  PROC DrawPart176()
    MoveL Offs(pOrigin,258.82,201.40,0.00),v40,fine,tPen\WObj:=wPaper;
    MoveL Offs(pOrigin,258.82,201.40,6.00),v60,z5,tPen\WObj:=wPaper;
    MoveL Offs(pOrigin,257.32,201.40,6.00),vTravel,z5,tPen\WObj:=wPaper;
    MoveL Offs(pOrigin,257.32,201.40,0.00),v60,z0,tPen\WObj:=wPaper;
    MoveL Offs(pOrigin,259.12,199.60,0.00),v40,fine,tPen\WObj:=wPaper;
    MoveL Offs(pOrigin,259.12,199.60,6.00),v60,z5,tPen\WObj:=wPaper;
    MoveL Offs(pOrigin,257.63,199.61,6.00),vTravel,z5,tPen\WObj:=wPaper;
    MoveL Offs(pOrigin,257.63,199.61,0.00),v60,z0,tPen\WObj:=wPaper;
    MoveL Offs(pOrigin,255.52,201.71,0.00),v40,fine,tPen\WObj:=wPaper;
    MoveL Offs(pOrigin,255.52,201.71,6.00),v60,z5,tPen\WObj:=wPaper;
    MoveL Offs(pOrigin,253.72,202.01,6.00),vTravel,z5,tPen\WObj:=wPaper;
    MoveL Offs(pOrigin,253.72,202.01,0.00),v60,z0,tPen\WObj:=wPaper;
    MoveL Offs(pOrigin,255.98,199.76,0.00),v40,fine,tPen\WObj:=wPaper;
    MoveL Offs(pOrigin,255.98,199.76,6.00),v60,z5,tPen\WObj:=wPaper;
    MoveL Offs(pOrigin,254.48,199.77,6.00),vTravel,z5,tPen\WObj:=wPaper;
    MoveL Offs(pOrigin,254.48,199.77,0.00),v60,z0,tPen\WObj:=wPaper;
    MoveL Offs(pOrigin,252.23,202.02,0.00),v40,z0,tPen\WObj:=wPaper;
    MoveL Offs(pOrigin,251.94,201.46,0.00),v40,z0,tPen\WObj:=wPaper;
    MoveL Offs(pOrigin,251.19,200.71,0.00),v40,z0,tPen\WObj:=wPaper;
    MoveL Offs(pOrigin,251.33,199.92,0.00),v40,z0,tPen\WObj:=wPaper;
    MoveL Offs(pOrigin,249.53,201.73,0.00),v40,fine,tPen\WObj:=wPaper;
    MoveL Offs(pOrigin,249.53,201.73,6.00),v60,z5,tPen\WObj:=wPaper;
    MoveL Offs(pOrigin,250.73,202.02,6.00),vTravel,z5,tPen\WObj:=wPaper;
    MoveL Offs(pOrigin,250.73,202.02,0.00),v60,z0,tPen\WObj:=wPaper;
    MoveL Offs(pOrigin,252.98,199.77,0.00),v40,fine,tPen\WObj:=wPaper;
    MoveL Offs(pOrigin,252.98,199.77,6.00),v60,z5,tPen\WObj:=wPaper;
    MoveL Offs(pOrigin,251.76,206.96,6.00),vTravel,z5,tPen\WObj:=wPaper;
    MoveL Offs(pOrigin,251.76,206.96,0.00),v60,z0,tPen\WObj:=wPaper;
    MoveL Offs(pOrigin,249.06,209.67,0.00),v40,z0,tPen\WObj:=wPaper;
    MoveL Offs(pOrigin,249.42,209.39,0.00),v40,z0,tPen\WObj:=wPaper;
    MoveL Offs(pOrigin,247.16,207.14,0.00),v40,z0,tPen\WObj:=wPaper;
    MoveL Offs(pOrigin,247.57,206.68,0.00),v40,z0,tPen\WObj:=wPaper;
    MoveL Offs(pOrigin,245.01,209.23,0.00),v40,z0,tPen\WObj:=wPaper;
    MoveL Offs(pOrigin,244.47,208.93,0.00),v40,z0,tPen\WObj:=wPaper;
    MoveL Offs(pOrigin,242.67,207.12,0.00),v40,z0,tPen\WObj:=wPaper;
    MoveL Offs(pOrigin,243.07,206.69,0.00),v40,z0,tPen\WObj:=wPaper;
    MoveL Offs(pOrigin,240.37,209.40,0.00),v40,z0,tPen\WObj:=wPaper;
    MoveL Offs(pOrigin,239.98,208.91,0.00),v40,z0,tPen\WObj:=wPaper;
    MoveL Offs(pOrigin,238.78,207.71,0.00),v40,z0,tPen\WObj:=wPaper;
    MoveL Offs(pOrigin,238.10,208.15,0.00),v40,z0,tPen\WObj:=wPaper;
    MoveL Offs(pOrigin,240.86,207.51,0.00),v40,z0,tPen\WObj:=wPaper;
    MoveL Offs(pOrigin,248.30,207.51,0.00),v40,z0,tPen\WObj:=wPaper;
    MoveL Offs(pOrigin,256.16,208.79,0.00),v40,z0,tPen\WObj:=wPaper;
    MoveL Offs(pOrigin,259.14,209.71,0.00),v40,z0,tPen\WObj:=wPaper;
    MoveL Offs(pOrigin,259.56,210.49,0.00),v40,z0,tPen\WObj:=wPaper;
    MoveL Offs(pOrigin,259.56,210.49,0.00),v40,z0,tPen\WObj:=wPaper;
    MoveL Offs(pOrigin,253.61,209.21,0.00),v40,z0,tPen\WObj:=wPaper;
    MoveL Offs(pOrigin,247.24,208.36,0.00),v40,z0,tPen\WObj:=wPaper;
    MoveL Offs(pOrigin,241.07,208.36,0.00),v40,z0,tPen\WObj:=wPaper;
    MoveL Offs(pOrigin,238.10,208.79,0.00),v40,z0,tPen\WObj:=wPaper;
    MoveL Offs(pOrigin,238.10,208.79,0.00),v40,z0,tPen\WObj:=wPaper;
    MoveL Offs(pOrigin,237.04,209.00,0.00),v40,z0,tPen\WObj:=wPaper;
    MoveL Offs(pOrigin,237.04,209.00,0.00),v40,z0,tPen\WObj:=wPaper;
    MoveL Offs(pOrigin,237.46,208.15,0.00),v40,z0,tPen\WObj:=wPaper;
    MoveL Offs(pOrigin,237.89,208.15,0.00),v40,z0,tPen\WObj:=wPaper;
    MoveL Offs(pOrigin,238.10,208.79,0.00),v40,z0,tPen\WObj:=wPaper;
    MoveL Offs(pOrigin,238.63,209.06,0.00),v40,z0,tPen\WObj:=wPaper;
    MoveL Offs(pOrigin,237.58,208.01,0.00),v40,z0,tPen\WObj:=wPaper;
    MoveL Offs(pOrigin,237.04,209.00,0.00),v40,z0,tPen\WObj:=wPaper;
    MoveL Offs(pOrigin,234.49,209.35,0.00),v40,z0,tPen\WObj:=wPaper;
    MoveL Offs(pOrigin,232.15,210.70,0.00),v40,z0,tPen\WObj:=wPaper;
    MoveL Offs(pOrigin,231.51,210.91,0.00),v40,z0,tPen\WObj:=wPaper;
    MoveL Offs(pOrigin,230.45,212.12,0.00),v40,z0,tPen\WObj:=wPaper;
    MoveL Offs(pOrigin,227.26,214.52,0.00),v40,fine,tPen\WObj:=wPaper;
    MoveL Offs(pOrigin,227.26,214.52,6.00),v60,z5,tPen\WObj:=wPaper;
    MoveL Offs(pOrigin,228.97,213.33,6.00),vTravel,z5,tPen\WObj:=wPaper;
    MoveL Offs(pOrigin,228.97,213.33,0.00),v60,z0,tPen\WObj:=wPaper;
    MoveL Offs(pOrigin,234.08,208.22,0.00),v40,z0,tPen\WObj:=wPaper;
    MoveL Offs(pOrigin,234.29,209.19,0.00),v40,z0,tPen\WObj:=wPaper;
    MoveL Offs(pOrigin,235.04,209.94,0.00),v40,z0,tPen\WObj:=wPaper;
    MoveL Offs(pOrigin,233.99,210.39,0.00),v40,z0,tPen\WObj:=wPaper;
    MoveL Offs(pOrigin,233.24,209.64,0.00),v40,fine,tPen\WObj:=wPaper;
    MoveL Offs(pOrigin,233.24,209.64,6.00),v60,z5,tPen\WObj:=wPaper;
    MoveL Offs(pOrigin,234.07,211.21,6.00),vTravel,z5,tPen\WObj:=wPaper;
    MoveL Offs(pOrigin,234.07,211.21,0.00),v60,z0,tPen\WObj:=wPaper;
    MoveL Offs(pOrigin,238.28,207.01,0.00),v40,fine,tPen\WObj:=wPaper;
    MoveL Offs(pOrigin,238.28,207.01,6.00),v60,z5,tPen\WObj:=wPaper;
    MoveL Offs(pOrigin,239.93,206.85,6.00),vTravel,z5,tPen\WObj:=wPaper;
    MoveL Offs(pOrigin,239.93,206.85,0.00),v60,z0,tPen\WObj:=wPaper;
    MoveL Offs(pOrigin,236.47,210.31,0.00),v40,z0,tPen\WObj:=wPaper;
    MoveL Offs(pOrigin,236.39,209.80,0.00),v40,z0,tPen\WObj:=wPaper;
    MoveL Offs(pOrigin,235.19,208.60,0.00),v40,z0,tPen\WObj:=wPaper;
    MoveL Offs(pOrigin,236.23,208.15,0.00),v40,z0,tPen\WObj:=wPaper;
    MoveL Offs(pOrigin,237.43,209.35,0.00),v40,z0,tPen\WObj:=wPaper;
    MoveL Offs(pOrigin,238.57,209.70,0.00),v40,z0,tPen\WObj:=wPaper;
    MoveL Offs(pOrigin,241.58,206.70,0.00),v40,z0,tPen\WObj:=wPaper;
    MoveL Offs(pOrigin,241.47,207.42,0.00),v40,z0,tPen\WObj:=wPaper;
    MoveL Offs(pOrigin,242.98,208.92,0.00),v40,z0,tPen\WObj:=wPaper;
    MoveL Offs(pOrigin,243.52,209.24,0.00),v40,z0,tPen\WObj:=wPaper;
    MoveL Offs(pOrigin,246.07,206.68,0.00),v40,z0,tPen\WObj:=wPaper;
    MoveL Offs(pOrigin,245.67,207.13,0.00),v40,z0,tPen\WObj:=wPaper;
    MoveL Offs(pOrigin,247.62,209.08,0.00),v40,z0,tPen\WObj:=wPaper;
    MoveL Offs(pOrigin,247.86,209.37,0.00),v40,z0,tPen\WObj:=wPaper;
    MoveL Offs(pOrigin,250.41,206.82,0.00),v40,z0,tPen\WObj:=wPaper;
    MoveL Offs(pOrigin,250.61,207.60,0.00),v40,z0,tPen\WObj:=wPaper;
    MoveL Offs(pOrigin,252.87,209.85,0.00),v40,z0,tPen\WObj:=wPaper;
    MoveL Offs(pOrigin,253.10,210.11,0.00),v40,z0,tPen\WObj:=wPaper;
    MoveL Offs(pOrigin,255.50,207.70,0.00),v40,z0,tPen\WObj:=wPaper;
    MoveL Offs(pOrigin,255.86,208.36,0.00),v40,z0,tPen\WObj:=wPaper;
    MoveL Offs(pOrigin,258.26,210.77,0.00),v40,z0,tPen\WObj:=wPaper;
    MoveL Offs(pOrigin,258.04,211.14,0.00),v40,z0,tPen\WObj:=wPaper;
    MoveL Offs(pOrigin,260.14,209.04,0.00),v40,z0,tPen\WObj:=wPaper;
    MoveL Offs(pOrigin,260.06,209.57,0.00),v40,z0,tPen\WObj:=wPaper;
    MoveL Offs(pOrigin,263.36,212.88,0.00),v40,z0,tPen\WObj:=wPaper;
    MoveL Offs(pOrigin,263.28,213.37,0.00),v40,z0,tPen\WObj:=wPaper;
    MoveL Offs(pOrigin,265.08,211.57,0.00),v40,z0,tPen\WObj:=wPaper;
    MoveL Offs(pOrigin,264.45,212.40,0.00),v40,z0,tPen\WObj:=wPaper;
    MoveL Offs(pOrigin,265.73,212.19,0.00),v40,z0,tPen\WObj:=wPaper;
    MoveL Offs(pOrigin,265.94,212.82,0.00),v40,z0,tPen\WObj:=wPaper;
    MoveL Offs(pOrigin,265.83,212.31,0.00),v40,z0,tPen\WObj:=wPaper;
    MoveL Offs(pOrigin,264.32,213.82,0.00),v40,z0,tPen\WObj:=wPaper;
    MoveL Offs(pOrigin,265.22,214.41,0.00),v40,z0,tPen\WObj:=wPaper;
    MoveL Offs(pOrigin,266.72,212.91,0.00),v40,z0,tPen\WObj:=wPaper;
    MoveL Offs(pOrigin,267.32,213.81,0.00),v40,z0,tPen\WObj:=wPaper;
    MoveL Offs(pOrigin,265.97,215.16,0.00),v40,z0,tPen\WObj:=wPaper;
    MoveL Offs(pOrigin,266.36,214.39,0.00),v40,z0,tPen\WObj:=wPaper;
    MoveL Offs(pOrigin,262.60,210.63,0.00),v40,z0,tPen\WObj:=wPaper;
    MoveL Offs(pOrigin,263.29,210.37,0.00),v40,z0,tPen\WObj:=wPaper;
    MoveL Offs(pOrigin,261.33,212.33,0.00),v40,z0,tPen\WObj:=wPaper;
    MoveL Offs(pOrigin,262.38,212.77,0.00),v40,z0,tPen\WObj:=wPaper;
  ENDPROC

  PROC DrawPart177()
    MoveL Offs(pOrigin,264.18,210.97,0.00),v40,fine,tPen\WObj:=wPaper;
    MoveL Offs(pOrigin,264.18,210.97,6.00),v60,z5,tPen\WObj:=wPaper;
    MoveL Offs(pOrigin,264.45,212.40,6.00),vTravel,z5,tPen\WObj:=wPaper;
    MoveL Offs(pOrigin,264.45,212.40,0.00),v60,z0,tPen\WObj:=wPaper;
    MoveL Offs(pOrigin,262.33,211.20,0.00),v40,z0,tPen\WObj:=wPaper;
    MoveL Offs(pOrigin,259.56,210.49,0.00),v40,z0,tPen\WObj:=wPaper;
    MoveL Offs(pOrigin,259.24,211.44,0.00),v40,z0,tPen\WObj:=wPaper;
    MoveL Offs(pOrigin,261.19,209.48,0.00),v40,z0,tPen\WObj:=wPaper;
    MoveL Offs(pOrigin,262.24,209.93,0.00),v40,z0,tPen\WObj:=wPaper;
    MoveL Offs(pOrigin,260.29,211.88,0.00),v40,z0,tPen\WObj:=wPaper;
    MoveL Offs(pOrigin,260.36,211.37,0.00),v40,z0,tPen\WObj:=wPaper;
    MoveL Offs(pOrigin,257.96,208.97,0.00),v40,z0,tPen\WObj:=wPaper;
    MoveL Offs(pOrigin,257.90,208.29,0.00),v40,z0,tPen\WObj:=wPaper;
    MoveL Offs(pOrigin,255.65,210.55,0.00),v40,z0,tPen\WObj:=wPaper;
    MoveL Offs(pOrigin,256.46,210.46,0.00),v40,z0,tPen\WObj:=wPaper;
    MoveL Offs(pOrigin,254.21,208.21,0.00),v40,z0,tPen\WObj:=wPaper;
    MoveL Offs(pOrigin,254.31,207.41,0.00),v40,z0,tPen\WObj:=wPaper;
    MoveL Offs(pOrigin,251.60,210.11,0.00),v40,z0,tPen\WObj:=wPaper;
    MoveL Offs(pOrigin,251.07,209.54,0.00),v40,z0,tPen\WObj:=wPaper;
    MoveL Offs(pOrigin,248.96,207.44,0.00),v40,z0,tPen\WObj:=wPaper;
    MoveL Offs(pOrigin,248.92,206.82,0.00),v40,z0,tPen\WObj:=wPaper;
    MoveL Offs(pOrigin,246.51,209.23,0.00),v40,z0,tPen\WObj:=wPaper;
    MoveL Offs(pOrigin,245.97,208.93,0.00),v40,z0,tPen\WObj:=wPaper;
    MoveL Offs(pOrigin,244.17,207.13,0.00),v40,z0,tPen\WObj:=wPaper;
    MoveL Offs(pOrigin,244.57,206.69,0.00),v40,z0,tPen\WObj:=wPaper;
    MoveL Offs(pOrigin,242.02,209.24,0.00),v40,z0,tPen\WObj:=wPaper;
    MoveL Offs(pOrigin,241.48,208.92,0.00),v40,z0,tPen\WObj:=wPaper;
    MoveL Offs(pOrigin,240.13,207.56,0.00),v40,fine,tPen\WObj:=wPaper;
    MoveL Offs(pOrigin,240.13,207.56,6.00),v60,z5,tPen\WObj:=wPaper;
    MoveL Offs(pOrigin,236.48,207.31,6.00),vTravel,z5,tPen\WObj:=wPaper;
    MoveL Offs(pOrigin,236.48,207.31,0.00),v60,z0,tPen\WObj:=wPaper;
    MoveL Offs(pOrigin,231.22,212.57,0.00),v40,fine,tPen\WObj:=wPaper;
    MoveL Offs(pOrigin,231.22,212.57,6.00),v60,z5,tPen\WObj:=wPaper;
    MoveL Offs(pOrigin,229.60,208.36,6.00),vTravel,z5,tPen\WObj:=wPaper;
    MoveL Offs(pOrigin,229.60,208.36,0.00),v60,z0,tPen\WObj:=wPaper;
    MoveL Offs(pOrigin,227.90,208.72,0.00),v40,z0,tPen\WObj:=wPaper;
    MoveL Offs(pOrigin,222.16,210.98,0.00),v40,z0,tPen\WObj:=wPaper;
    MoveL Offs(pOrigin,215.15,217.29,0.00),v40,z0,tPen\WObj:=wPaper;
    MoveL Offs(pOrigin,211.89,221.75,0.00),v40,z0,tPen\WObj:=wPaper;
    MoveL Offs(pOrigin,209.98,225.57,0.00),v40,z0,tPen\WObj:=wPaper;
    MoveL Offs(pOrigin,207.93,232.38,0.00),v40,z0,tPen\WObj:=wPaper;
    MoveL Offs(pOrigin,207.29,232.38,0.00),v40,z0,tPen\WObj:=wPaper;
    MoveL Offs(pOrigin,207.07,233.44,0.00),v40,z0,tPen\WObj:=wPaper;
    MoveL Offs(pOrigin,207.29,233.65,0.00),v40,z0,tPen\WObj:=wPaper;
    MoveL Offs(pOrigin,206.29,233.02,0.00),v40,z0,tPen\WObj:=wPaper;
    MoveL Offs(pOrigin,209.30,230.01,0.00),v40,z0,tPen\WObj:=wPaper;
    MoveL Offs(pOrigin,208.74,229.94,0.00),v40,z0,tPen\WObj:=wPaper;
    MoveL Offs(pOrigin,205.73,226.93,0.00),v40,z0,tPen\WObj:=wPaper;
    MoveL Offs(pOrigin,206.01,227.26,0.00),v40,z0,tPen\WObj:=wPaper;
    MoveL Offs(pOrigin,209.20,227.26,0.00),v40,z0,tPen\WObj:=wPaper;
    MoveL Offs(pOrigin,209.92,226.65,0.00),v40,z0,tPen\WObj:=wPaper;
    MoveL Offs(pOrigin,208.42,225.14,0.00),v40,z0,tPen\WObj:=wPaper;
    MoveL Offs(pOrigin,208.99,225.14,0.00),v40,z0,tPen\WObj:=wPaper;
    MoveL Offs(pOrigin,210.05,225.14,0.00),v40,z0,tPen\WObj:=wPaper;
    MoveL Offs(pOrigin,209.62,226.20,0.00),v40,z0,tPen\WObj:=wPaper;
    MoveL Offs(pOrigin,208.56,226.20,0.00),v40,z0,tPen\WObj:=wPaper;
    MoveL Offs(pOrigin,208.05,227.28,0.00),v40,z0,tPen\WObj:=wPaper;
    MoveL Offs(pOrigin,208.05,228.34,0.00),v40,fine,tPen\WObj:=wPaper;
    MoveL Offs(pOrigin,208.05,228.34,6.00),v60,z5,tPen\WObj:=wPaper;
    MoveL Offs(pOrigin,205.71,226.13,6.00),vTravel,z5,tPen\WObj:=wPaper;
    MoveL Offs(pOrigin,205.71,226.13,0.00),v60,z0,tPen\WObj:=wPaper;
    MoveL Offs(pOrigin,201.81,230.04,0.00),v40,z0,tPen\WObj:=wPaper;
    MoveL Offs(pOrigin,202.74,229.92,0.00),v40,z0,tPen\WObj:=wPaper;
    MoveL Offs(pOrigin,204.25,231.42,0.00),v40,z0,tPen\WObj:=wPaper;
    MoveL Offs(pOrigin,204.65,231.68,0.00),v40,z0,tPen\WObj:=wPaper;
    MoveL Offs(pOrigin,201.19,235.13,0.00),v40,z0,tPen\WObj:=wPaper;
    MoveL Offs(pOrigin,202.19,234.65,0.00),v40,z0,tPen\WObj:=wPaper;
    MoveL Offs(pOrigin,203.46,234.65,0.00),v40,z0,tPen\WObj:=wPaper;
    MoveL Offs(pOrigin,203.81,233.97,0.00),v40,z0,tPen\WObj:=wPaper;
    MoveL Offs(pOrigin,201.85,232.01,0.00),v40,z0,tPen\WObj:=wPaper;
    MoveL Offs(pOrigin,201.76,232.54,0.00),v40,z0,tPen\WObj:=wPaper;
    MoveL Offs(pOrigin,203.46,232.54,0.00),v40,z0,tPen\WObj:=wPaper;
    MoveL Offs(pOrigin,202.77,232.80,0.00),v40,z0,tPen\WObj:=wPaper;
    MoveL Offs(pOrigin,202.77,234.08,0.00),v40,z0,tPen\WObj:=wPaper;
    MoveL Offs(pOrigin,203.46,233.59,0.00),v40,z0,tPen\WObj:=wPaper;
    MoveL Offs(pOrigin,201.34,233.59,0.00),v40,fine,tPen\WObj:=wPaper;
    MoveL Offs(pOrigin,201.34,233.59,6.00),v60,z5,tPen\WObj:=wPaper;
    MoveL Offs(pOrigin,200.52,238.15,6.00),vTravel,z5,tPen\WObj:=wPaper;
    MoveL Offs(pOrigin,200.52,238.15,0.00),v60,z0,tPen\WObj:=wPaper;
    MoveL Offs(pOrigin,203.08,240.71,0.00),v40,z0,tPen\WObj:=wPaper;
    MoveL Offs(pOrigin,202.61,239.93,0.00),v40,z0,tPen\WObj:=wPaper;
    MoveL Offs(pOrigin,200.06,239.93,0.00),v40,fine,tPen\WObj:=wPaper;
    MoveL Offs(pOrigin,200.06,239.93,6.00),v60,z5,tPen\WObj:=wPaper;
    MoveL Offs(pOrigin,199.34,244.44,6.00),vTravel,z5,tPen\WObj:=wPaper;
    MoveL Offs(pOrigin,199.34,244.44,0.00),v60,z0,tPen\WObj:=wPaper;
    MoveL Offs(pOrigin,201.00,246.09,0.00),v40,fine,tPen\WObj:=wPaper;
    MoveL Offs(pOrigin,201.00,246.09,6.00),v60,z5,tPen\WObj:=wPaper;
    MoveL Offs(pOrigin,202.80,246.96,6.00),vTravel,z5,tPen\WObj:=wPaper;
    MoveL Offs(pOrigin,202.80,246.96,0.00),v60,z0,tPen\WObj:=wPaper;
    MoveL Offs(pOrigin,194.24,255.53,0.00),v40,z0,tPen\WObj:=wPaper;
    MoveL Offs(pOrigin,194.59,256.11,0.00),v40,z0,tPen\WObj:=wPaper;
    MoveL Offs(pOrigin,196.39,257.91,0.00),v40,fine,tPen\WObj:=wPaper;
    MoveL Offs(pOrigin,196.39,257.91,6.00),v60,z5,tPen\WObj:=wPaper;
    MoveL Offs(pOrigin,196.38,256.41,6.00),vTravel,z5,tPen\WObj:=wPaper;
    MoveL Offs(pOrigin,196.38,256.41,0.00),v60,z0,tPen\WObj:=wPaper;
    MoveL Offs(pOrigin,194.58,254.61,0.00),v40,z0,tPen\WObj:=wPaper;
    MoveL Offs(pOrigin,194.24,254.03,0.00),v40,z0,tPen\WObj:=wPaper;
    MoveL Offs(pOrigin,207.47,240.80,0.00),v40,z0,tPen\WObj:=wPaper;
    MoveL Offs(pOrigin,206.65,241.51,0.00),v40,z0,tPen\WObj:=wPaper;
    MoveL Offs(pOrigin,206.86,242.79,0.00),v40,z0,tPen\WObj:=wPaper;
    MoveL Offs(pOrigin,206.44,243.21,0.00),v40,z0,tPen\WObj:=wPaper;
    MoveL Offs(pOrigin,206.44,243.21,0.00),v40,z0,tPen\WObj:=wPaper;
    MoveL Offs(pOrigin,206.86,245.98,0.00),v40,z0,tPen\WObj:=wPaper;
    MoveL Offs(pOrigin,206.65,248.10,0.00),v40,z0,tPen\WObj:=wPaper;
    MoveL Offs(pOrigin,207.14,247.76,0.00),v40,z0,tPen\WObj:=wPaper;
    MoveL Offs(pOrigin,206.39,247.01,0.00),v40,fine,tPen\WObj:=wPaper;
    MoveL Offs(pOrigin,206.39,247.01,6.00),v60,z5,tPen\WObj:=wPaper;
    MoveL Offs(pOrigin,207.75,246.50,6.00),vTravel,z5,tPen\WObj:=wPaper;
    MoveL Offs(pOrigin,207.75,246.50,0.00),v60,z0,tPen\WObj:=wPaper;
    MoveL Offs(pOrigin,204.29,249.95,0.00),v40,z0,tPen\WObj:=wPaper;
    MoveL Offs(pOrigin,204.90,250.00,0.00),v40,z0,tPen\WObj:=wPaper;
    MoveL Offs(pOrigin,207.31,252.40,0.00),v40,z0,tPen\WObj:=wPaper;
    MoveL Offs(pOrigin,206.86,252.60,0.00),v40,z0,tPen\WObj:=wPaper;
    MoveL Offs(pOrigin,204.52,252.60,0.00),v40,z0,tPen\WObj:=wPaper;
    MoveL Offs(pOrigin,204.31,252.39,0.00),v40,z0,tPen\WObj:=wPaper;
    MoveL Offs(pOrigin,208.37,256.45,0.00),v40,z0,tPen\WObj:=wPaper;
    MoveL Offs(pOrigin,208.91,257.28,0.00),v40,z0,tPen\WObj:=wPaper;
    MoveL Offs(pOrigin,195.69,270.50,0.00),v40,z0,tPen\WObj:=wPaper;
    MoveL Offs(pOrigin,196.45,270.41,0.00),v40,z0,tPen\WObj:=wPaper;
    MoveL Offs(pOrigin,196.24,270.84,0.00),v40,z0,tPen\WObj:=wPaper;
  ENDPROC

  PROC DrawPart178()
    MoveL Offs(pOrigin,196.45,270.41,0.00),v40,z0,tPen\WObj:=wPaper;
    MoveL Offs(pOrigin,196.73,270.20,0.00),v40,z0,tPen\WObj:=wPaper;
    MoveL Offs(pOrigin,204.54,278.01,0.00),v40,z0,tPen\WObj:=wPaper;
    MoveL Offs(pOrigin,205.55,278.56,0.00),v40,z0,tPen\WObj:=wPaper;
    MoveL Offs(pOrigin,189.03,295.09,0.00),v40,z0,tPen\WObj:=wPaper;
    MoveL Offs(pOrigin,189.91,294.74,0.00),v40,z0,tPen\WObj:=wPaper;
    MoveL Offs(pOrigin,197.57,302.41,0.00),v40,z0,tPen\WObj:=wPaper;
    MoveL Offs(pOrigin,198.36,302.50,0.00),v40,z0,tPen\WObj:=wPaper;
    MoveL Offs(pOrigin,198.79,302.36,0.00),v40,z0,tPen\WObj:=wPaper;
    MoveL Offs(pOrigin,200.70,303.14,0.00),v40,z0,tPen\WObj:=wPaper;
    MoveL Offs(pOrigin,201.34,302.92,0.00),v40,z0,tPen\WObj:=wPaper;
    MoveL Offs(pOrigin,200.72,302.57,0.00),v40,z0,tPen\WObj:=wPaper;
    MoveL Offs(pOrigin,210.04,311.88,0.00),v40,z0,tPen\WObj:=wPaper;
    MoveL Offs(pOrigin,210.26,311.85,0.00),v40,z0,tPen\WObj:=wPaper;
    MoveL Offs(pOrigin,210.05,312.06,0.00),v40,z0,tPen\WObj:=wPaper;
    MoveL Offs(pOrigin,210.69,311.42,0.00),v40,z0,tPen\WObj:=wPaper;
    MoveL Offs(pOrigin,211.75,311.42,0.00),v40,z0,tPen\WObj:=wPaper;
    MoveL Offs(pOrigin,212.60,311.74,0.00),v40,z0,tPen\WObj:=wPaper;
    MoveL Offs(pOrigin,226.84,311.74,0.00),v40,z0,tPen\WObj:=wPaper;
    MoveL Offs(pOrigin,226.84,312.79,0.00),v40,z0,tPen\WObj:=wPaper;
    MoveL Offs(pOrigin,225.14,312.79,0.00),v40,z0,tPen\WObj:=wPaper;
    MoveL Offs(pOrigin,224.50,312.91,0.00),v40,z0,tPen\WObj:=wPaper;
    MoveL Offs(pOrigin,223.86,313.34,0.00),v40,z0,tPen\WObj:=wPaper;
    MoveL Offs(pOrigin,223.86,313.76,0.00),v40,z0,tPen\WObj:=wPaper;
    MoveL Offs(pOrigin,223.01,313.76,0.00),v40,z0,tPen\WObj:=wPaper;
    MoveL Offs(pOrigin,222.59,314.61,0.00),v40,z0,tPen\WObj:=wPaper;
    MoveL Offs(pOrigin,222.38,316.52,0.00),v40,z0,tPen\WObj:=wPaper;
    MoveL Offs(pOrigin,221.60,316.95,0.00),v40,z0,tPen\WObj:=wPaper;
    MoveL Offs(pOrigin,221.52,317.59,0.00),v40,z0,tPen\WObj:=wPaper;
    MoveL Offs(pOrigin,223.30,320.35,0.00),v40,z0,tPen\WObj:=wPaper;
    MoveL Offs(pOrigin,224.07,322.48,0.00),v40,z0,tPen\WObj:=wPaper;
    MoveL Offs(pOrigin,224.07,322.48,0.00),v40,z0,tPen\WObj:=wPaper;
    MoveL Offs(pOrigin,224.78,323.11,0.00),v40,z0,tPen\WObj:=wPaper;
    MoveL Offs(pOrigin,225.14,324.17,0.00),v40,z0,tPen\WObj:=wPaper;
    MoveL Offs(pOrigin,224.93,327.79,0.00),v40,z0,tPen\WObj:=wPaper;
    MoveL Offs(pOrigin,224.77,328.10,0.00),v40,z0,tPen\WObj:=wPaper;
    MoveL Offs(pOrigin,225.67,329.01,0.00),v40,z0,tPen\WObj:=wPaper;
    MoveL Offs(pOrigin,224.71,329.06,0.00),v40,z0,tPen\WObj:=wPaper;
    MoveL Offs(pOrigin,223.86,331.19,0.00),v40,z0,tPen\WObj:=wPaper;
    MoveL Offs(pOrigin,223.86,331.19,0.00),v40,z0,tPen\WObj:=wPaper;
    MoveL Offs(pOrigin,222.38,331.61,0.00),v40,z0,tPen\WObj:=wPaper;
    MoveL Offs(pOrigin,219.40,331.40,0.00),v40,z0,tPen\WObj:=wPaper;
    MoveL Offs(pOrigin,217.70,331.68,0.00),v40,z0,tPen\WObj:=wPaper;
    MoveL Offs(pOrigin,217.49,332.04,0.00),v40,z0,tPen\WObj:=wPaper;
    MoveL Offs(pOrigin,217.29,331.08,0.00),v40,z0,tPen\WObj:=wPaper;
    MoveL Offs(pOrigin,225.25,339.04,0.00),v40,z0,tPen\WObj:=wPaper;
    MoveL Offs(pOrigin,225.59,339.17,0.00),v40,z0,tPen\WObj:=wPaper;
    MoveL Offs(pOrigin,230.70,334.06,0.00),v40,z0,tPen\WObj:=wPaper;
    MoveL Offs(pOrigin,231.38,334.72,0.00),v40,z0,tPen\WObj:=wPaper;
    MoveL Offs(pOrigin,233.18,336.52,0.00),v40,z0,tPen\WObj:=wPaper;
    MoveL Offs(pOrigin,232.64,336.60,0.00),v40,z0,tPen\WObj:=wPaper;
    MoveL Offs(pOrigin,241.50,327.73,0.00),v40,z0,tPen\WObj:=wPaper;
    MoveL Offs(pOrigin,241.09,328.01,0.00),v40,z0,tPen\WObj:=wPaper;
    MoveL Offs(pOrigin,223.06,309.97,0.00),v40,z0,tPen\WObj:=wPaper;
    MoveL Offs(pOrigin,224.03,309.36,0.00),v40,z0,tPen\WObj:=wPaper;
    MoveL Offs(pOrigin,211.71,321.68,0.00),v40,z0,tPen\WObj:=wPaper;
    MoveL Offs(pOrigin,211.86,321.17,0.00),v40,z0,tPen\WObj:=wPaper;
    MoveL Offs(pOrigin,210.06,319.37,0.00),v40,z0,tPen\WObj:=wPaper;
    MoveL Offs(pOrigin,210.90,319.71,0.00),v40,z0,tPen\WObj:=wPaper;
    MoveL Offs(pOrigin,209.41,320.14,0.00),v40,z0,tPen\WObj:=wPaper;
    MoveL Offs(pOrigin,209.31,320.12,0.00),v40,z0,tPen\WObj:=wPaper;
    MoveL Offs(pOrigin,210.82,321.62,0.00),v40,z0,tPen\WObj:=wPaper;
    MoveL Offs(pOrigin,209.77,322.07,0.00),v40,z0,tPen\WObj:=wPaper;
    MoveL Offs(pOrigin,208.42,320.71,0.00),v40,z0,tPen\WObj:=wPaper;
    MoveL Offs(pOrigin,207.52,321.31,0.00),v40,z0,tPen\WObj:=wPaper;
    MoveL Offs(pOrigin,208.87,322.66,0.00),v40,fine,tPen\WObj:=wPaper;
    MoveL Offs(pOrigin,208.87,322.66,6.00),v60,z5,tPen\WObj:=wPaper;
    MoveL Offs(pOrigin,207.52,322.81,6.00),vTravel,z5,tPen\WObj:=wPaper;
    MoveL Offs(pOrigin,207.52,322.81,0.00),v60,z0,tPen\WObj:=wPaper;
    MoveL Offs(pOrigin,205.12,320.40,0.00),v40,fine,tPen\WObj:=wPaper;
    MoveL Offs(pOrigin,205.12,320.40,6.00),v60,z5,tPen\WObj:=wPaper;
    MoveL Offs(pOrigin,204.10,322.30,6.00),vTravel,z5,tPen\WObj:=wPaper;
    MoveL Offs(pOrigin,204.10,322.30,0.00),v60,z0,tPen\WObj:=wPaper;
    MoveL Offs(pOrigin,201.12,322.30,0.00),v40,z0,tPen\WObj:=wPaper;
    MoveL Offs(pOrigin,200.18,322.77,0.00),v40,z0,tPen\WObj:=wPaper;
    MoveL Offs(pOrigin,216.70,306.24,0.00),v40,z0,tPen\WObj:=wPaper;
    MoveL Offs(pOrigin,216.85,306.54,0.00),v40,z0,tPen\WObj:=wPaper;
    MoveL Offs(pOrigin,215.79,305.05,0.00),v40,z0,tPen\WObj:=wPaper;
    MoveL Offs(pOrigin,214.94,305.12,0.00),v40,z0,tPen\WObj:=wPaper;
    MoveL Offs(pOrigin,214.30,305.90,0.00),v40,z0,tPen\WObj:=wPaper;
    MoveL Offs(pOrigin,214.30,305.90,0.00),v40,z0,tPen\WObj:=wPaper;
    MoveL Offs(pOrigin,214.73,306.54,0.00),v40,z0,tPen\WObj:=wPaper;
    MoveL Offs(pOrigin,216.85,306.96,0.00),v40,z0,tPen\WObj:=wPaper;
    MoveL Offs(pOrigin,216.00,307.51,0.00),v40,z0,tPen\WObj:=wPaper;
    MoveL Offs(pOrigin,200.06,307.51,0.00),v40,z0,tPen\WObj:=wPaper;
    MoveL Offs(pOrigin,199.62,308.39,0.00),v40,z0,tPen\WObj:=wPaper;
    MoveL Offs(pOrigin,209.84,298.17,0.00),v40,z0,tPen\WObj:=wPaper;
    MoveL Offs(pOrigin,209.24,297.27,0.00),v40,z0,tPen\WObj:=wPaper;
    MoveL Offs(pOrigin,198.42,308.09,0.00),v40,z0,tPen\WObj:=wPaper;
    MoveL Offs(pOrigin,198.49,307.80,0.00),v40,z0,tPen\WObj:=wPaper;
    MoveL Offs(pOrigin,190.53,299.84,0.00),v40,fine,tPen\WObj:=wPaper;
    MoveL Offs(pOrigin,190.53,299.84,6.00),v60,z5,tPen\WObj:=wPaper;
    MoveL Offs(pOrigin,190.82,298.64,6.00),vTravel,z5,tPen\WObj:=wPaper;
    MoveL Offs(pOrigin,190.82,298.64,0.00),v60,z0,tPen\WObj:=wPaper;
    MoveL Offs(pOrigin,200.59,308.41,0.00),v40,z0,tPen\WObj:=wPaper;
    MoveL Offs(pOrigin,200.67,308.83,0.00),v40,z0,tPen\WObj:=wPaper;
    MoveL Offs(pOrigin,209.98,299.52,0.00),v40,z0,tPen\WObj:=wPaper;
    MoveL Offs(pOrigin,210.73,300.27,0.00),v40,z0,tPen\WObj:=wPaper;
    MoveL Offs(pOrigin,201.71,309.28,0.00),v40,z0,tPen\WObj:=wPaper;
    MoveL Offs(pOrigin,201.34,309.94,0.00),v40,z0,tPen\WObj:=wPaper;
    MoveL Offs(pOrigin,203.04,309.73,0.00),v40,z0,tPen\WObj:=wPaper;
    MoveL Offs(pOrigin,204.31,310.58,0.00),v40,z0,tPen\WObj:=wPaper;
    MoveL Offs(pOrigin,204.49,310.82,0.00),v40,z0,tPen\WObj:=wPaper;
    MoveL Offs(pOrigin,205.24,311.57,0.00),v40,z0,tPen\WObj:=wPaper;
    MoveL Offs(pOrigin,206.29,311.12,0.00),v40,z0,tPen\WObj:=wPaper;
    MoveL Offs(pOrigin,201.63,306.46,0.00),v40,fine,tPen\WObj:=wPaper;
    MoveL Offs(pOrigin,201.63,306.46,6.00),v60,z5,tPen\WObj:=wPaper;
    MoveL Offs(pOrigin,201.93,305.27,6.00),vTravel,z5,tPen\WObj:=wPaper;
    MoveL Offs(pOrigin,201.93,305.27,0.00),v60,z0,tPen\WObj:=wPaper;
    MoveL Offs(pOrigin,199.67,303.01,0.00),v40,fine,tPen\WObj:=wPaper;
    MoveL Offs(pOrigin,199.67,303.01,6.00),v60,z5,tPen\WObj:=wPaper;
    MoveL Offs(pOrigin,199.33,304.19,6.00),vTravel,z5,tPen\WObj:=wPaper;
    MoveL Offs(pOrigin,199.33,304.19,0.00),v60,z0,tPen\WObj:=wPaper;
    MoveL Offs(pOrigin,208.35,295.18,0.00),v40,z0,tPen\WObj:=wPaper;
    MoveL Offs(pOrigin,208.80,296.23,0.00),v40,z0,tPen\WObj:=wPaper;
    MoveL Offs(pOrigin,193.62,311.40,0.00),v40,z0,tPen\WObj:=wPaper;
    MoveL Offs(pOrigin,194.32,310.68,0.00),v40,z0,tPen\WObj:=wPaper;
    MoveL Offs(pOrigin,196.24,310.68,0.00),v40,z0,tPen\WObj:=wPaper;
    MoveL Offs(pOrigin,196.45,311.74,0.00),v40,z0,tPen\WObj:=wPaper;
    MoveL Offs(pOrigin,194.75,311.74,0.00),v40,z0,tPen\WObj:=wPaper;
  ENDPROC

  PROC DrawPart179()
    MoveL Offs(pOrigin,194.07,312.45,0.00),v40,z0,tPen\WObj:=wPaper;
    MoveL Offs(pOrigin,197.52,308.99,0.00),v40,z0,tPen\WObj:=wPaper;
    MoveL Offs(pOrigin,198.12,309.89,0.00),v40,z0,tPen\WObj:=wPaper;
    MoveL Offs(pOrigin,194.51,313.50,0.00),v40,fine,tPen\WObj:=wPaper;
    MoveL Offs(pOrigin,194.51,313.50,6.00),v60,z5,tPen\WObj:=wPaper;
    MoveL Offs(pOrigin,196.43,312.70,6.00),vTravel,z5,tPen\WObj:=wPaper;
    MoveL Offs(pOrigin,196.43,312.70,0.00),v60,z0,tPen\WObj:=wPaper;
    MoveL Offs(pOrigin,196.43,314.40,0.00),v40,z0,tPen\WObj:=wPaper;
    MoveL Offs(pOrigin,196.24,314.90,0.00),v40,z0,tPen\WObj:=wPaper;
    MoveL Offs(pOrigin,200.49,314.90,0.00),v40,z0,tPen\WObj:=wPaper;
    MoveL Offs(pOrigin,199.60,315.04,0.00),v40,z0,tPen\WObj:=wPaper;
    MoveL Offs(pOrigin,199.60,316.52,0.00),v40,z0,tPen\WObj:=wPaper;
    MoveL Offs(pOrigin,199.42,317.02,0.00),v40,z0,tPen\WObj:=wPaper;
    MoveL Offs(pOrigin,206.65,317.02,0.00),v40,z0,tPen\WObj:=wPaper;
    MoveL Offs(pOrigin,206.60,315.92,0.00),v40,z0,tPen\WObj:=wPaper;
    MoveL Offs(pOrigin,208.26,317.57,0.00),v40,z0,tPen\WObj:=wPaper;
    MoveL Offs(pOrigin,207.83,318.10,0.00),v40,z0,tPen\WObj:=wPaper;
    MoveL Offs(pOrigin,218.65,307.28,0.00),v40,fine,tPen\WObj:=wPaper;
    MoveL Offs(pOrigin,218.65,307.28,6.00),v60,z5,tPen\WObj:=wPaper;
    MoveL Offs(pOrigin,217.49,308.02,6.00),vTravel,z5,tPen\WObj:=wPaper;
    MoveL Offs(pOrigin,217.49,308.02,0.00),v60,z0,tPen\WObj:=wPaper;
    MoveL Offs(pOrigin,215.57,308.52,0.00),v40,z0,tPen\WObj:=wPaper;
    MoveL Offs(pOrigin,214.94,309.16,0.00),v40,z0,tPen\WObj:=wPaper;
    MoveL Offs(pOrigin,214.51,308.88,0.00),v40,z0,tPen\WObj:=wPaper;
    MoveL Offs(pOrigin,214.38,308.66,0.00),v40,z0,tPen\WObj:=wPaper;
    MoveL Offs(pOrigin,214.38,307.39,0.00),v40,z0,tPen\WObj:=wPaper;
    MoveL Offs(pOrigin,214.30,306.46,0.00),v40,z0,tPen\WObj:=wPaper;
    MoveL Offs(pOrigin,204.74,306.46,0.00),v40,z0,tPen\WObj:=wPaper;
    MoveL Offs(pOrigin,204.74,306.11,0.00),v40,z0,tPen\WObj:=wPaper;
    MoveL Offs(pOrigin,203.68,306.33,0.00),v40,z0,tPen\WObj:=wPaper;
    MoveL Offs(pOrigin,203.25,306.75,0.00),v40,z0,tPen\WObj:=wPaper;
    MoveL Offs(pOrigin,202.83,306.17,0.00),v40,z0,tPen\WObj:=wPaper;
    MoveL Offs(pOrigin,207.64,310.98,0.00),v40,z0,tPen\WObj:=wPaper;
    MoveL Offs(pOrigin,208.14,312.06,0.00),v40,z0,tPen\WObj:=wPaper;
    MoveL Offs(pOrigin,208.56,311.85,0.00),v40,z0,tPen\WObj:=wPaper;
    MoveL Offs(pOrigin,208.14,312.06,0.00),v40,fine,tPen\WObj:=wPaper;
    MoveL Offs(pOrigin,208.14,312.06,6.00),v60,z5,tPen\WObj:=wPaper;
    MoveL Offs(pOrigin,209.84,312.06,6.00),vTravel,z5,tPen\WObj:=wPaper;
    MoveL Offs(pOrigin,209.84,312.06,0.00),v60,z0,tPen\WObj:=wPaper;
    MoveL Offs(pOrigin,207.93,313.41,0.00),v40,z0,tPen\WObj:=wPaper;
    MoveL Offs(pOrigin,206.65,313.55,0.00),v40,fine,tPen\WObj:=wPaper;
    MoveL Offs(pOrigin,206.65,313.55,6.00),v60,z5,tPen\WObj:=wPaper;
    MoveL Offs(pOrigin,205.90,312.56,6.00),vTravel,z5,tPen\WObj:=wPaper;
    MoveL Offs(pOrigin,205.90,312.56,0.00),v60,z0,tPen\WObj:=wPaper;
    MoveL Offs(pOrigin,214.16,304.30,0.00),v40,z0,tPen\WObj:=wPaper;
    MoveL Offs(pOrigin,214.91,305.05,0.00),v40,z0,tPen\WObj:=wPaper;
    MoveL Offs(pOrigin,198.68,321.27,0.00),v40,z0,tPen\WObj:=wPaper;
    MoveL Offs(pOrigin,199.64,321.62,0.00),v40,z0,tPen\WObj:=wPaper;
    MoveL Offs(pOrigin,200.49,322.48,0.00),v40,z0,tPen\WObj:=wPaper;
    MoveL Offs(pOrigin,199.64,321.62,0.00),v40,z0,tPen\WObj:=wPaper;
    MoveL Offs(pOrigin,199.43,322.02,0.00),v40,z0,tPen\WObj:=wPaper;
    MoveL Offs(pOrigin,215.81,305.64,0.00),v40,fine,tPen\WObj:=wPaper;
    MoveL Offs(pOrigin,215.81,305.64,6.00),v60,z5,tPen\WObj:=wPaper;
    MoveL Offs(pOrigin,214.06,305.45,6.00),vTravel,z5,tPen\WObj:=wPaper;
    MoveL Offs(pOrigin,214.06,305.45,0.00),v60,z0,tPen\WObj:=wPaper;
    MoveL Offs(pOrigin,233.60,324.99,0.00),v40,z0,tPen\WObj:=wPaper;
    MoveL Offs(pOrigin,232.57,324.60,0.00),v40,z0,tPen\WObj:=wPaper;
    MoveL Offs(pOrigin,232.79,325.02,0.00),v40,z0,tPen\WObj:=wPaper;
    MoveL Offs(pOrigin,232.57,324.60,0.00),v40,fine,tPen\WObj:=wPaper;
    MoveL Offs(pOrigin,232.57,324.60,6.00),v60,z5,tPen\WObj:=wPaper;
    MoveL Offs(pOrigin,232.52,326.26,6.00),vTravel,z5,tPen\WObj:=wPaper;
    MoveL Offs(pOrigin,232.52,326.26,0.00),v60,z0,tPen\WObj:=wPaper;
    MoveL Offs(pOrigin,246.65,312.14,0.00),v40,z0,tPen\WObj:=wPaper;
    MoveL Offs(pOrigin,247.39,312.89,0.00),v40,z0,tPen\WObj:=wPaper;
    MoveL Offs(pOrigin,235.22,325.06,0.00),v40,z0,tPen\WObj:=wPaper;
    MoveL Offs(pOrigin,235.82,325.95,0.00),v40,z0,tPen\WObj:=wPaper;
    MoveL Offs(pOrigin,249.79,311.98,0.00),v40,z0,tPen\WObj:=wPaper;
    MoveL Offs(pOrigin,249.79,311.21,0.00),v40,z0,tPen\WObj:=wPaper;
    MoveL Offs(pOrigin,249.50,312.49,0.00),v40,z0,tPen\WObj:=wPaper;
    MoveL Offs(pOrigin,250.43,315.25,0.00),v40,z0,tPen\WObj:=wPaper;
    MoveL Offs(pOrigin,251.06,315.46,0.00),v40,z0,tPen\WObj:=wPaper;
    MoveL Offs(pOrigin,251.06,315.46,0.00),v40,z0,tPen\WObj:=wPaper;
    MoveL Offs(pOrigin,251.27,316.31,0.00),v40,z0,tPen\WObj:=wPaper;
    MoveL Offs(pOrigin,252.34,317.16,0.00),v40,z0,tPen\WObj:=wPaper;
    MoveL Offs(pOrigin,252.34,317.16,0.00),v40,z0,tPen\WObj:=wPaper;
    MoveL Offs(pOrigin,255.31,318.01,0.00),v40,z0,tPen\WObj:=wPaper;
    MoveL Offs(pOrigin,255.31,318.01,0.00),v40,z0,tPen\WObj:=wPaper;
    MoveL Offs(pOrigin,256.16,318.44,0.00),v40,z0,tPen\WObj:=wPaper;
    MoveL Offs(pOrigin,255.31,318.01,0.00),v40,z0,tPen\WObj:=wPaper;
    MoveL Offs(pOrigin,254.82,315.67,0.00),v40,z0,tPen\WObj:=wPaper;
    MoveL Offs(pOrigin,252.98,313.55,0.00),v40,z0,tPen\WObj:=wPaper;
    MoveL Offs(pOrigin,252.55,312.49,0.00),v40,z0,tPen\WObj:=wPaper;
    MoveL Offs(pOrigin,252.55,312.49,0.00),v40,z0,tPen\WObj:=wPaper;
    MoveL Offs(pOrigin,251.70,312.42,0.00),v40,z0,tPen\WObj:=wPaper;
    MoveL Offs(pOrigin,250.92,313.12,0.00),v40,z0,tPen\WObj:=wPaper;
    MoveL Offs(pOrigin,251.06,315.46,0.00),v40,z0,tPen\WObj:=wPaper;
    MoveL Offs(pOrigin,251.28,314.90,0.00),v40,z0,tPen\WObj:=wPaper;
    MoveL Offs(pOrigin,257.44,314.90,0.00),v40,z0,tPen\WObj:=wPaper;
    MoveL Offs(pOrigin,258.08,315.04,0.00),v40,z0,tPen\WObj:=wPaper;
    MoveL Offs(pOrigin,257.79,314.19,0.00),v40,z0,tPen\WObj:=wPaper;
    MoveL Offs(pOrigin,256.66,313.12,0.00),v40,z0,tPen\WObj:=wPaper;
    MoveL Offs(pOrigin,255.81,311.42,0.00),v40,z0,tPen\WObj:=wPaper;
    MoveL Offs(pOrigin,255.74,310.58,0.00),v40,z0,tPen\WObj:=wPaper;
    MoveL Offs(pOrigin,255.74,310.58,0.00),v40,z0,tPen\WObj:=wPaper;
    MoveL Offs(pOrigin,257.23,311.85,0.00),v40,z0,tPen\WObj:=wPaper;
    MoveL Offs(pOrigin,259.77,313.34,0.00),v40,z0,tPen\WObj:=wPaper;
    MoveL Offs(pOrigin,259.77,313.34,0.00),v40,z0,tPen\WObj:=wPaper;
    MoveL Offs(pOrigin,265.94,314.68,0.00),v40,z0,tPen\WObj:=wPaper;
    MoveL Offs(pOrigin,266.15,315.89,0.00),v40,z0,tPen\WObj:=wPaper;
    MoveL Offs(pOrigin,266.15,315.89,0.00),v40,z0,tPen\WObj:=wPaper;
    MoveL Offs(pOrigin,270.61,316.74,0.00),v40,z0,tPen\WObj:=wPaper;
    MoveL Offs(pOrigin,272.10,316.52,0.00),v40,z0,tPen\WObj:=wPaper;
    MoveL Offs(pOrigin,274.23,316.95,0.00),v40,z0,tPen\WObj:=wPaper;
    MoveL Offs(pOrigin,274.46,316.57,0.00),v40,z0,tPen\WObj:=wPaper;
    MoveL Offs(pOrigin,266.80,308.91,0.00),v40,z0,tPen\WObj:=wPaper;
    MoveL Offs(pOrigin,265.94,309.30,0.00),v40,z0,tPen\WObj:=wPaper;
    MoveL Offs(pOrigin,267.00,308.66,0.00),v40,z0,tPen\WObj:=wPaper;
    MoveL Offs(pOrigin,268.49,308.59,0.00),v40,z0,tPen\WObj:=wPaper;
    MoveL Offs(pOrigin,269.34,308.02,0.00),v40,z0,tPen\WObj:=wPaper;
    MoveL Offs(pOrigin,272.74,307.60,0.00),v40,z0,tPen\WObj:=wPaper;
    MoveL Offs(pOrigin,272.46,306.75,0.00),v40,z0,tPen\WObj:=wPaper;
    MoveL Offs(pOrigin,272.46,308.66,0.00),v40,z0,tPen\WObj:=wPaper;
    MoveL Offs(pOrigin,273.52,308.66,0.00),v40,z0,tPen\WObj:=wPaper;
    MoveL Offs(pOrigin,273.52,306.32,0.00),v40,z0,tPen\WObj:=wPaper;
    MoveL Offs(pOrigin,273.59,305.69,0.00),v40,z0,tPen\WObj:=wPaper;
    MoveL Offs(pOrigin,270.40,306.75,0.00),v40,z0,tPen\WObj:=wPaper;
    MoveL Offs(pOrigin,270.40,306.75,0.00),v40,z0,tPen\WObj:=wPaper;
    MoveL Offs(pOrigin,269.34,307.81,0.00),v40,z0,tPen\WObj:=wPaper;
    MoveL Offs(pOrigin,268.70,307.39,0.00),v40,z0,tPen\WObj:=wPaper;
    MoveL Offs(pOrigin,268.70,307.39,0.00),v40,z0,tPen\WObj:=wPaper;
  ENDPROC

  PROC DrawPart180()
    MoveL Offs(pOrigin,265.30,307.67,0.00),v40,z0,tPen\WObj:=wPaper;
    MoveL Offs(pOrigin,265.09,308.66,0.00),v40,z0,tPen\WObj:=wPaper;
    MoveL Offs(pOrigin,265.09,308.66,0.00),v40,z0,tPen\WObj:=wPaper;
    MoveL Offs(pOrigin,265.94,309.30,0.00),v40,z0,tPen\WObj:=wPaper;
    MoveL Offs(pOrigin,265.90,309.51,0.00),v40,z0,tPen\WObj:=wPaper;
    MoveL Offs(pOrigin,274.17,317.77,0.00),v40,z0,tPen\WObj:=wPaper;
    MoveL Offs(pOrigin,274.65,317.16,0.00),v40,z0,tPen\WObj:=wPaper;
    MoveL Offs(pOrigin,276.14,317.59,0.00),v40,fine,tPen\WObj:=wPaper;
    MoveL Offs(pOrigin,276.14,317.59,6.00),v60,z5,tPen\WObj:=wPaper;
    MoveL Offs(pOrigin,276.43,319.69,6.00),vTravel,z5,tPen\WObj:=wPaper;
    MoveL Offs(pOrigin,276.43,319.69,0.00),v60,z0,tPen\WObj:=wPaper;
    MoveL Offs(pOrigin,275.38,320.74,0.00),v40,z0,tPen\WObj:=wPaper;
    MoveL Offs(pOrigin,275.71,320.35,0.00),v40,z0,tPen\WObj:=wPaper;
    MoveL Offs(pOrigin,275.29,319.29,0.00),v40,z0,tPen\WObj:=wPaper;
    MoveL Offs(pOrigin,274.65,319.08,0.00),v40,z0,tPen\WObj:=wPaper;
    MoveL Offs(pOrigin,274.44,319.50,0.00),v40,fine,tPen\WObj:=wPaper;
    MoveL Offs(pOrigin,274.44,319.50,6.00),v60,z5,tPen\WObj:=wPaper;
    MoveL Offs(pOrigin,272.69,320.45,6.00),vTravel,z5,tPen\WObj:=wPaper;
    MoveL Offs(pOrigin,272.69,320.45,0.00),v60,z0,tPen\WObj:=wPaper;
    MoveL Offs(pOrigin,282.15,310.98,0.00),v40,z0,tPen\WObj:=wPaper;
    MoveL Offs(pOrigin,283.05,311.58,0.00),v40,z0,tPen\WObj:=wPaper;
    MoveL Offs(pOrigin,278.09,316.54,0.00),v40,z0,tPen\WObj:=wPaper;
    MoveL Offs(pOrigin,277.91,315.53,0.00),v40,z0,tPen\WObj:=wPaper;
    MoveL Offs(pOrigin,269.49,307.12,0.00),v40,z0,tPen\WObj:=wPaper;
    MoveL Offs(pOrigin,268.70,307.39,0.00),v40,z0,tPen\WObj:=wPaper;
    MoveL Offs(pOrigin,269.12,305.97,0.00),v40,z0,tPen\WObj:=wPaper;
    MoveL Offs(pOrigin,269.98,305.97,0.00),v40,z0,tPen\WObj:=wPaper;
    MoveL Offs(pOrigin,270.40,306.75,0.00),v40,z0,tPen\WObj:=wPaper;
    MoveL Offs(pOrigin,270.54,306.67,0.00),v40,z0,tPen\WObj:=wPaper;
    MoveL Offs(pOrigin,276.40,312.53,0.00),v40,fine,tPen\WObj:=wPaper;
    MoveL Offs(pOrigin,276.40,312.53,6.00),v60,z5,tPen\WObj:=wPaper;
    MoveL Offs(pOrigin,276.77,313.85,6.00),vTravel,z5,tPen\WObj:=wPaper;
    MoveL Offs(pOrigin,276.77,313.85,0.00),v60,z0,tPen\WObj:=wPaper;
    MoveL Offs(pOrigin,273.80,313.85,0.00),v40,z0,tPen\WObj:=wPaper;
    MoveL Offs(pOrigin,274.31,314.92,0.00),v40,z0,tPen\WObj:=wPaper;
    MoveL Offs(pOrigin,267.85,308.46,0.00),v40,z0,tPen\WObj:=wPaper;
    MoveL Offs(pOrigin,268.75,307.87,0.00),v40,z0,tPen\WObj:=wPaper;
    MoveL Offs(pOrigin,276.26,315.38,0.00),v40,fine,tPen\WObj:=wPaper;
    MoveL Offs(pOrigin,276.26,315.38,6.00),v60,z5,tPen\WObj:=wPaper;
    MoveL Offs(pOrigin,277.62,315.25,6.00),vTravel,z5,tPen\WObj:=wPaper;
    MoveL Offs(pOrigin,277.62,315.25,0.00),v60,z0,tPen\WObj:=wPaper;
    MoveL Offs(pOrigin,278.26,316.10,0.00),v40,z0,tPen\WObj:=wPaper;
    MoveL Offs(pOrigin,279.54,316.31,0.00),v40,z0,tPen\WObj:=wPaper;
    MoveL Offs(pOrigin,279.44,316.68,0.00),v40,z0,tPen\WObj:=wPaper;
    MoveL Offs(pOrigin,280.34,315.78,0.00),v40,z0,tPen\WObj:=wPaper;
    MoveL Offs(pOrigin,280.81,316.52,0.00),v40,z0,tPen\WObj:=wPaper;
    MoveL Offs(pOrigin,281.24,317.16,0.00),v40,z0,tPen\WObj:=wPaper;
    MoveL Offs(pOrigin,282.30,317.16,0.00),v40,z0,tPen\WObj:=wPaper;
    MoveL Offs(pOrigin,282.30,317.16,0.00),v40,z0,tPen\WObj:=wPaper;
    MoveL Offs(pOrigin,283.36,317.38,0.00),v40,z0,tPen\WObj:=wPaper;
    MoveL Offs(pOrigin,283.36,317.38,0.00),v40,z0,tPen\WObj:=wPaper;
    MoveL Offs(pOrigin,283.15,316.52,0.00),v40,z0,tPen\WObj:=wPaper;
    MoveL Offs(pOrigin,282.51,316.52,0.00),v40,z0,tPen\WObj:=wPaper;
    MoveL Offs(pOrigin,282.30,317.16,0.00),v40,z0,tPen\WObj:=wPaper;
    MoveL Offs(pOrigin,282.30,316.52,0.00),v40,z0,tPen\WObj:=wPaper;
    MoveL Offs(pOrigin,281.02,316.31,0.00),v40,z0,tPen\WObj:=wPaper;
    MoveL Offs(pOrigin,280.81,316.52,0.00),v40,z0,tPen\WObj:=wPaper;
    MoveL Offs(pOrigin,280.81,316.52,0.00),v40,z0,tPen\WObj:=wPaper;
    MoveL Offs(pOrigin,279.54,316.10,0.00),v40,z0,tPen\WObj:=wPaper;
    MoveL Offs(pOrigin,278.69,314.83,0.00),v40,z0,tPen\WObj:=wPaper;
    MoveL Offs(pOrigin,278.69,314.83,0.00),v40,z0,tPen\WObj:=wPaper;
    MoveL Offs(pOrigin,278.69,315.04,0.00),v40,z0,tPen\WObj:=wPaper;
    MoveL Offs(pOrigin,278.48,314.83,0.00),v40,z0,tPen\WObj:=wPaper;
    MoveL Offs(pOrigin,279.33,314.19,0.00),v40,z0,tPen\WObj:=wPaper;
    MoveL Offs(pOrigin,279.54,313.55,0.00),v40,z0,tPen\WObj:=wPaper;
    MoveL Offs(pOrigin,279.25,312.39,0.00),v40,z0,tPen\WObj:=wPaper;
    MoveL Offs(pOrigin,272.33,305.48,0.00),v40,z0,tPen\WObj:=wPaper;
    MoveL Offs(pOrigin,272.31,304.62,0.00),v40,z0,tPen\WObj:=wPaper;
    MoveL Offs(pOrigin,271.89,305.05,0.00),v40,z0,tPen\WObj:=wPaper;
    MoveL Offs(pOrigin,270.61,305.26,0.00),v40,z0,tPen\WObj:=wPaper;
    MoveL Offs(pOrigin,270.19,305.90,0.00),v40,fine,tPen\WObj:=wPaper;
    MoveL Offs(pOrigin,270.19,305.90,6.00),v60,z5,tPen\WObj:=wPaper;
    MoveL Offs(pOrigin,268.98,306.23,6.00),vTravel,z5,tPen\WObj:=wPaper;
    MoveL Offs(pOrigin,268.98,306.23,0.00),v60,z0,tPen\WObj:=wPaper;
    MoveL Offs(pOrigin,248.70,326.51,0.00),v40,fine,tPen\WObj:=wPaper;
    MoveL Offs(pOrigin,248.70,326.51,6.00),v60,z5,tPen\WObj:=wPaper;
    MoveL Offs(pOrigin,249.48,327.43,6.00),vTravel,z5,tPen\WObj:=wPaper;
    MoveL Offs(pOrigin,249.48,327.43,0.00),v60,z0,tPen\WObj:=wPaper;
    MoveL Offs(pOrigin,250.83,328.78,0.00),v40,fine,tPen\WObj:=wPaper;
    MoveL Offs(pOrigin,250.83,328.78,6.00),v60,z5,tPen\WObj:=wPaper;
    MoveL Offs(pOrigin,250.38,326.84,6.00),vTravel,z5,tPen\WObj:=wPaper;
    MoveL Offs(pOrigin,250.38,326.84,0.00),v60,z0,tPen\WObj:=wPaper;
    MoveL Offs(pOrigin,236.70,313.16,0.00),v40,fine,tPen\WObj:=wPaper;
    MoveL Offs(pOrigin,236.70,313.16,6.00),v60,z5,tPen\WObj:=wPaper;
    MoveL Offs(pOrigin,237.25,312.06,6.00),vTravel,z5,tPen\WObj:=wPaper;
    MoveL Offs(pOrigin,237.25,312.06,0.00),v60,z0,tPen\WObj:=wPaper;
    MoveL Offs(pOrigin,238.17,310.36,0.00),v40,z0,tPen\WObj:=wPaper;
    MoveL Offs(pOrigin,238.74,310.15,0.00),v40,z0,tPen\WObj:=wPaper;
    MoveL Offs(pOrigin,238.74,310.15,0.00),v40,z0,tPen\WObj:=wPaper;
    MoveL Offs(pOrigin,239.59,310.79,0.00),v40,z0,tPen\WObj:=wPaper;
    MoveL Offs(pOrigin,239.76,310.06,0.00),v40,z0,tPen\WObj:=wPaper;
    MoveL Offs(pOrigin,221.58,328.24,0.00),v40,z0,tPen\WObj:=wPaper;
    MoveL Offs(pOrigin,221.47,327.80,0.00),v40,z0,tPen\WObj:=wPaper;
    MoveL Offs(pOrigin,220.72,327.04,0.00),v40,z0,tPen\WObj:=wPaper;
    MoveL Offs(pOrigin,220.27,328.09,0.00),v40,z0,tPen\WObj:=wPaper;
    MoveL Offs(pOrigin,219.07,326.89,0.00),v40,z0,tPen\WObj:=wPaper;
    MoveL Offs(pOrigin,218.76,326.73,0.00),v40,z0,tPen\WObj:=wPaper;
    MoveL Offs(pOrigin,220.04,325.88,0.00),v40,z0,tPen\WObj:=wPaper;
    MoveL Offs(pOrigin,220.25,325.24,0.00),v40,z0,tPen\WObj:=wPaper;
    MoveL Offs(pOrigin,220.68,325.24,0.00),v40,z0,tPen\WObj:=wPaper;
    MoveL Offs(pOrigin,220.68,325.24,0.00),v40,z0,tPen\WObj:=wPaper;
    MoveL Offs(pOrigin,221.95,325.66,0.00),v40,z0,tPen\WObj:=wPaper;
    MoveL Offs(pOrigin,221.95,325.66,0.00),v40,z0,tPen\WObj:=wPaper;
    MoveL Offs(pOrigin,222.59,325.24,0.00),v40,z0,tPen\WObj:=wPaper;
    MoveL Offs(pOrigin,222.59,323.11,0.00),v40,z0,tPen\WObj:=wPaper;
    MoveL Offs(pOrigin,221.95,322.26,0.00),v40,z0,tPen\WObj:=wPaper;
    MoveL Offs(pOrigin,221.95,322.26,0.00),v40,z0,tPen\WObj:=wPaper;
    MoveL Offs(pOrigin,220.75,324.17,0.00),v40,z0,tPen\WObj:=wPaper;
    MoveL Offs(pOrigin,220.68,325.24,0.00),v40,fine,tPen\WObj:=wPaper;
    MoveL Offs(pOrigin,220.68,325.24,6.00),v60,z5,tPen\WObj:=wPaper;
    MoveL Offs(pOrigin,220.68,323.96,6.00),vTravel,z5,tPen\WObj:=wPaper;
    MoveL Offs(pOrigin,220.68,323.96,0.00),v60,z0,tPen\WObj:=wPaper;
    MoveL Offs(pOrigin,220.46,321.84,0.00),v40,z0,tPen\WObj:=wPaper;
    MoveL Offs(pOrigin,219.80,321.65,0.00),v40,z0,tPen\WObj:=wPaper;
    MoveL Offs(pOrigin,217.25,319.09,0.00),v40,z0,tPen\WObj:=wPaper;
    MoveL Offs(pOrigin,216.81,319.57,0.00),v40,z0,tPen\WObj:=wPaper;
    MoveL Offs(pOrigin,226.58,309.80,0.00),v40,z0,tPen\WObj:=wPaper;
    MoveL Offs(pOrigin,226.84,309.30,0.00),v40,z0,tPen\WObj:=wPaper;
    MoveL Offs(pOrigin,225.56,310.36,0.00),v40,z0,tPen\WObj:=wPaper;
    MoveL Offs(pOrigin,224.07,310.15,0.00),v40,z0,tPen\WObj:=wPaper;
  ENDPROC

  PROC DrawPart181()
    MoveL Offs(pOrigin,222.59,310.50,0.00),v40,z0,tPen\WObj:=wPaper;
    MoveL Offs(pOrigin,222.45,309.51,0.00),v40,z0,tPen\WObj:=wPaper;
    MoveL Offs(pOrigin,223.86,308.88,0.00),v40,fine,tPen\WObj:=wPaper;
    MoveL Offs(pOrigin,223.86,308.88,6.00),v60,z5,tPen\WObj:=wPaper;
    MoveL Offs(pOrigin,225.38,309.51,6.00),vTravel,z5,tPen\WObj:=wPaper;
    MoveL Offs(pOrigin,225.38,309.51,0.00),v60,z0,tPen\WObj:=wPaper;
    MoveL Offs(pOrigin,214.56,320.33,0.00),v40,fine,tPen\WObj:=wPaper;
    MoveL Offs(pOrigin,214.56,320.33,6.00),v60,z5,tPen\WObj:=wPaper;
    MoveL Offs(pOrigin,214.86,321.52,6.00),vTravel,z5,tPen\WObj:=wPaper;
    MoveL Offs(pOrigin,214.86,321.52,0.00),v60,z0,tPen\WObj:=wPaper;
    MoveL Offs(pOrigin,205.69,330.69,0.00),v40,z0,tPen\WObj:=wPaper;
    MoveL Offs(pOrigin,206.44,331.44,0.00),v40,z0,tPen\WObj:=wPaper;
    MoveL Offs(pOrigin,212.60,325.28,0.00),v40,fine,tPen\WObj:=wPaper;
    MoveL Offs(pOrigin,212.60,325.28,6.00),v60,z5,tPen\WObj:=wPaper;
    MoveL Offs(pOrigin,212.78,326.57,6.00),vTravel,z5,tPen\WObj:=wPaper;
    MoveL Offs(pOrigin,212.78,326.57,0.00),v60,z0,tPen\WObj:=wPaper;
    MoveL Offs(pOrigin,215.78,329.58,0.00),v40,z0,tPen\WObj:=wPaper;
    MoveL Offs(pOrigin,215.79,330.76,0.00),v40,z0,tPen\WObj:=wPaper;
    MoveL Offs(pOrigin,214.94,330.55,0.00),v40,z0,tPen\WObj:=wPaper;
    MoveL Offs(pOrigin,214.51,330.98,0.00),v40,z0,tPen\WObj:=wPaper;
    MoveL Offs(pOrigin,214.72,331.80,0.00),v40,z0,tPen\WObj:=wPaper;
    MoveL Offs(pOrigin,211.96,331.80,0.00),v40,z0,tPen\WObj:=wPaper;
    MoveL Offs(pOrigin,210.90,332.04,0.00),v40,z0,tPen\WObj:=wPaper;
    MoveL Offs(pOrigin,209.84,330.55,0.00),v40,z0,tPen\WObj:=wPaper;
    MoveL Offs(pOrigin,209.84,330.55,0.00),v40,z0,tPen\WObj:=wPaper;
    MoveL Offs(pOrigin,210.69,329.49,0.00),v40,z0,tPen\WObj:=wPaper;
    MoveL Offs(pOrigin,210.69,329.49,0.00),v40,z0,tPen\WObj:=wPaper;
    MoveL Offs(pOrigin,209.84,328.57,0.00),v40,z0,tPen\WObj:=wPaper;
    MoveL Offs(pOrigin,206.86,327.36,0.00),v40,z0,tPen\WObj:=wPaper;
    MoveL Offs(pOrigin,206.86,327.36,0.00),v40,z0,tPen\WObj:=wPaper;
    MoveL Offs(pOrigin,207.07,328.42,0.00),v40,z0,tPen\WObj:=wPaper;
    MoveL Offs(pOrigin,209.84,330.55,0.00),v40,z0,tPen\WObj:=wPaper;
    MoveL Offs(pOrigin,210.69,331.19,0.00),v40,z0,tPen\WObj:=wPaper;
    MoveL Offs(pOrigin,210.90,331.61,0.00),v40,z0,tPen\WObj:=wPaper;
    MoveL Offs(pOrigin,210.69,331.19,0.00),v40,z0,tPen\WObj:=wPaper;
    MoveL Offs(pOrigin,210.90,332.04,0.00),v40,z0,tPen\WObj:=wPaper;
    MoveL Offs(pOrigin,214.30,333.67,0.00),v40,z0,tPen\WObj:=wPaper;
    MoveL Offs(pOrigin,215.36,333.74,0.00),v40,z0,tPen\WObj:=wPaper;
    MoveL Offs(pOrigin,214.94,333.91,0.00),v40,z0,tPen\WObj:=wPaper;
    MoveL Offs(pOrigin,211.54,333.91,0.00),v40,z0,tPen\WObj:=wPaper;
    MoveL Offs(pOrigin,211.75,334.51,0.00),v40,z0,tPen\WObj:=wPaper;
    MoveL Offs(pOrigin,208.30,331.05,0.00),v40,z0,tPen\WObj:=wPaper;
    MoveL Offs(pOrigin,207.93,330.98,0.00),v40,z0,tPen\WObj:=wPaper;
    MoveL Offs(pOrigin,208.35,331.19,0.00),v40,z0,tPen\WObj:=wPaper;
    MoveL Offs(pOrigin,207.93,330.98,0.00),v40,z0,tPen\WObj:=wPaper;
    MoveL Offs(pOrigin,208.56,331.40,0.00),v40,z0,tPen\WObj:=wPaper;
    MoveL Offs(pOrigin,208.99,331.61,0.00),v40,z0,tPen\WObj:=wPaper;
    MoveL Offs(pOrigin,208.56,331.40,0.00),v40,fine,tPen\WObj:=wPaper;
    MoveL Offs(pOrigin,208.56,331.40,6.00),v60,z5,tPen\WObj:=wPaper;
    MoveL Offs(pOrigin,208.14,332.67,6.00),vTravel,z5,tPen\WObj:=wPaper;
    MoveL Offs(pOrigin,208.14,332.67,0.00),v60,z0,tPen\WObj:=wPaper;
    MoveL Offs(pOrigin,208.56,333.10,0.00),v40,z0,tPen\WObj:=wPaper;
    MoveL Offs(pOrigin,208.14,332.67,0.00),v40,z0,tPen\WObj:=wPaper;
    MoveL Offs(pOrigin,208.08,332.78,0.00),v40,z0,tPen\WObj:=wPaper;
    MoveL Offs(pOrigin,214.85,326.02,0.00),v40,z0,tPen\WObj:=wPaper;
    MoveL Offs(pOrigin,214.10,325.27,0.00),v40,z0,tPen\WObj:=wPaper;
    MoveL Offs(pOrigin,207.19,332.18,0.00),v40,fine,tPen\WObj:=wPaper;
    MoveL Offs(pOrigin,207.19,332.18,6.00),v60,z5,tPen\WObj:=wPaper;
    MoveL Offs(pOrigin,209.41,332.86,6.00),vTravel,z5,tPen\WObj:=wPaper;
    MoveL Offs(pOrigin,209.41,332.86,0.00),v60,z0,tPen\WObj:=wPaper;
    MoveL Offs(pOrigin,212.60,332.86,0.00),v40,fine,tPen\WObj:=wPaper;
    MoveL Offs(pOrigin,212.60,332.86,6.00),v60,z5,tPen\WObj:=wPaper;
    MoveL Offs(pOrigin,210.90,332.04,6.00),vTravel,z5,tPen\WObj:=wPaper;
    MoveL Offs(pOrigin,210.90,332.04,0.00),v60,z0,tPen\WObj:=wPaper;
    MoveL Offs(pOrigin,209.41,331.75,0.00),v40,z0,tPen\WObj:=wPaper;
    MoveL Offs(pOrigin,207.07,330.12,0.00),v40,z0,tPen\WObj:=wPaper;
    MoveL Offs(pOrigin,205.38,328.21,0.00),v40,z0,tPen\WObj:=wPaper;
    MoveL Offs(pOrigin,204.95,327.15,0.00),v40,z0,tPen\WObj:=wPaper;
    MoveL Offs(pOrigin,204.95,327.15,0.00),v40,z0,tPen\WObj:=wPaper;
    MoveL Offs(pOrigin,206.86,327.36,0.00),v40,z0,tPen\WObj:=wPaper;
    MoveL Offs(pOrigin,206.99,326.72,0.00),v40,z0,tPen\WObj:=wPaper;
    MoveL Offs(pOrigin,206.99,325.02,0.00),v40,z0,tPen\WObj:=wPaper;
    MoveL Offs(pOrigin,207.29,324.81,0.00),v40,z0,tPen\WObj:=wPaper;
    MoveL Offs(pOrigin,206.44,324.81,0.00),v40,z0,tPen\WObj:=wPaper;
    MoveL Offs(pOrigin,206.23,323.75,0.00),v40,z0,tPen\WObj:=wPaper;
    MoveL Offs(pOrigin,205.93,324.39,0.00),v40,z0,tPen\WObj:=wPaper;
    MoveL Offs(pOrigin,205.93,326.30,0.00),v40,z0,tPen\WObj:=wPaper;
    MoveL Offs(pOrigin,205.59,326.52,0.00),v40,z0,tPen\WObj:=wPaper;
    MoveL Offs(pOrigin,211.11,326.52,0.00),v40,z0,tPen\WObj:=wPaper;
    MoveL Offs(pOrigin,211.75,326.51,0.00),v40,z0,tPen\WObj:=wPaper;
    MoveL Offs(pOrigin,211.96,326.16,0.00),v40,z0,tPen\WObj:=wPaper;
    MoveL Offs(pOrigin,214.30,325.59,0.00),v40,z0,tPen\WObj:=wPaper;
    MoveL Offs(pOrigin,215.79,324.17,0.00),v40,fine,tPen\WObj:=wPaper;
    MoveL Offs(pOrigin,215.79,324.17,6.00),v60,z5,tPen\WObj:=wPaper;
    MoveL Offs(pOrigin,218.30,324.06,6.00),vTravel,z5,tPen\WObj:=wPaper;
    MoveL Offs(pOrigin,218.30,324.06,0.00),v60,z0,tPen\WObj:=wPaper;
    MoveL Offs(pOrigin,231.82,310.54,0.00),v40,fine,tPen\WObj:=wPaper;
    MoveL Offs(pOrigin,231.82,310.54,6.00),v60,z5,tPen\WObj:=wPaper;
    MoveL Offs(pOrigin,230.88,312.06,6.00),vTravel,z5,tPen\WObj:=wPaper;
    MoveL Offs(pOrigin,230.88,312.06,0.00),v60,z0,tPen\WObj:=wPaper;
    MoveL Offs(pOrigin,230.02,311.00,0.00),v40,z0,tPen\WObj:=wPaper;
    MoveL Offs(pOrigin,229.39,311.00,0.00),v40,z0,tPen\WObj:=wPaper;
    MoveL Offs(pOrigin,229.39,311.00,0.00),v40,z0,tPen\WObj:=wPaper;
    MoveL Offs(pOrigin,228.54,310.15,0.00),v40,z0,tPen\WObj:=wPaper;
    MoveL Offs(pOrigin,227.69,310.58,0.00),v40,z0,tPen\WObj:=wPaper;
    MoveL Offs(pOrigin,227.93,309.95,0.00),v40,z0,tPen\WObj:=wPaper;
    MoveL Offs(pOrigin,217.41,320.47,0.00),v40,z0,tPen\WObj:=wPaper;
    MoveL Offs(pOrigin,218.01,321.36,0.00),v40,z0,tPen\WObj:=wPaper;
    MoveL Offs(pOrigin,228.82,310.55,0.00),v40,z0,tPen\WObj:=wPaper;
    MoveL Offs(pOrigin,228.75,310.15,0.00),v40,z0,tPen\WObj:=wPaper;
    MoveL Offs(pOrigin,229.39,311.00,0.00),v40,z0,tPen\WObj:=wPaper;
    MoveL Offs(pOrigin,229.39,311.00,0.00),v40,z0,tPen\WObj:=wPaper;
    MoveL Offs(pOrigin,228.96,311.85,0.00),v40,z0,tPen\WObj:=wPaper;
    MoveL Offs(pOrigin,228.96,311.85,0.00),v40,z0,tPen\WObj:=wPaper;
    MoveL Offs(pOrigin,228.18,312.13,0.00),v40,z0,tPen\WObj:=wPaper;
    MoveL Offs(pOrigin,227.05,314.61,0.00),v40,z0,tPen\WObj:=wPaper;
    MoveL Offs(pOrigin,226.20,314.61,0.00),v40,z0,tPen\WObj:=wPaper;
    MoveL Offs(pOrigin,225.99,315.25,0.00),v40,z0,tPen\WObj:=wPaper;
    MoveL Offs(pOrigin,226.41,316.31,0.00),v40,z0,tPen\WObj:=wPaper;
    MoveL Offs(pOrigin,225.70,316.95,0.00),v40,z0,tPen\WObj:=wPaper;
    MoveL Offs(pOrigin,226.13,318.65,0.00),v40,z0,tPen\WObj:=wPaper;
    MoveL Offs(pOrigin,228.32,322.05,0.00),v40,z0,tPen\WObj:=wPaper;
    MoveL Offs(pOrigin,229.10,322.55,0.00),v40,z0,tPen\WObj:=wPaper;
    MoveL Offs(pOrigin,230.02,325.02,0.00),v40,z0,tPen\WObj:=wPaper;
    MoveL Offs(pOrigin,230.02,327.36,0.00),v40,z0,tPen\WObj:=wPaper;
    MoveL Offs(pOrigin,229.53,328.64,0.00),v40,z0,tPen\WObj:=wPaper;
    MoveL Offs(pOrigin,226.62,331.19,0.00),v40,z0,tPen\WObj:=wPaper;
    MoveL Offs(pOrigin,226.62,331.19,0.00),v40,z0,tPen\WObj:=wPaper;
    MoveL Offs(pOrigin,225.35,331.47,0.00),v40,z0,tPen\WObj:=wPaper;
    MoveL Offs(pOrigin,223.86,331.19,0.00),v40,z0,tPen\WObj:=wPaper;
  ENDPROC

  PROC DrawPart182()
    MoveL Offs(pOrigin,223.28,331.10,0.00),v40,z0,tPen\WObj:=wPaper;
    MoveL Offs(pOrigin,222.08,329.89,0.00),v40,z0,tPen\WObj:=wPaper;
    MoveL Offs(pOrigin,221.52,330.74,0.00),v40,z0,tPen\WObj:=wPaper;
    MoveL Offs(pOrigin,222.80,330.74,0.00),v40,z0,tPen\WObj:=wPaper;
    MoveL Offs(pOrigin,222.23,331.54,0.00),v40,z0,tPen\WObj:=wPaper;
    MoveL Offs(pOrigin,221.18,330.49,0.00),v40,z0,tPen\WObj:=wPaper;
    MoveL Offs(pOrigin,220.73,331.54,0.00),v40,z0,tPen\WObj:=wPaper;
    MoveL Offs(pOrigin,219.98,330.79,0.00),v40,z0,tPen\WObj:=wPaper;
    MoveL Offs(pOrigin,219.93,329.90,0.00),v40,z0,tPen\WObj:=wPaper;
    MoveL Offs(pOrigin,214.22,335.61,0.00),v40,z0,tPen\WObj:=wPaper;
    MoveL Offs(pOrigin,214.15,335.41,0.00),v40,z0,tPen\WObj:=wPaper;
    MoveL Offs(pOrigin,196.72,317.98,0.00),v40,z0,tPen\WObj:=wPaper;
    MoveL Offs(pOrigin,196.74,318.73,0.00),v40,z0,tPen\WObj:=wPaper;
    MoveL Offs(pOrigin,201.55,313.92,0.00),v40,fine,tPen\WObj:=wPaper;
    MoveL Offs(pOrigin,201.55,313.92,6.00),v60,z5,tPen\WObj:=wPaper;
    MoveL Offs(pOrigin,203.01,315.31,6.00),vTravel,z5,tPen\WObj:=wPaper;
    MoveL Offs(pOrigin,203.01,315.31,0.00),v60,z0,tPen\WObj:=wPaper;
    MoveL Offs(pOrigin,205.86,318.16,0.00),v40,fine,tPen\WObj:=wPaper;
    MoveL Offs(pOrigin,205.86,318.16,6.00),v60,z5,tPen\WObj:=wPaper;
    MoveL Offs(pOrigin,207.21,318.01,6.00),vTravel,z5,tPen\WObj:=wPaper;
    MoveL Offs(pOrigin,207.21,318.01,0.00),v60,z0,tPen\WObj:=wPaper;
    MoveL Offs(pOrigin,205.11,315.91,0.00),v40,z0,tPen\WObj:=wPaper;
    MoveL Offs(pOrigin,205.38,316.10,0.00),v40,z0,tPen\WObj:=wPaper;
    MoveL Offs(pOrigin,203.46,316.10,0.00),v40,z0,tPen\WObj:=wPaper;
    MoveL Offs(pOrigin,203.04,315.67,0.00),v40,z0,tPen\WObj:=wPaper;
    MoveL Offs(pOrigin,203.04,315.67,0.00),v40,z0,tPen\WObj:=wPaper;
    MoveL Offs(pOrigin,200.06,314.54,0.00),v40,z0,tPen\WObj:=wPaper;
    MoveL Offs(pOrigin,199.43,313.83,0.00),v40,z0,tPen\WObj:=wPaper;
    MoveL Offs(pOrigin,197.30,312.70,0.00),v40,z0,tPen\WObj:=wPaper;
    MoveL Offs(pOrigin,196.88,311.64,0.00),v40,fine,tPen\WObj:=wPaper;
    MoveL Offs(pOrigin,196.88,311.64,6.00),v60,z5,tPen\WObj:=wPaper;
    MoveL Offs(pOrigin,197.49,313.55,6.00),vTravel,z5,tPen\WObj:=wPaper;
    MoveL Offs(pOrigin,197.49,313.55,0.00),v60,z0,tPen\WObj:=wPaper;
    MoveL Offs(pOrigin,197.49,315.25,0.00),v40,z0,tPen\WObj:=wPaper;
    MoveL Offs(pOrigin,197.09,315.67,0.00),v40,z0,tPen\WObj:=wPaper;
    MoveL Offs(pOrigin,198.15,316.10,0.00),v40,z0,tPen\WObj:=wPaper;
    MoveL Offs(pOrigin,199.64,317.52,0.00),v40,z0,tPen\WObj:=wPaper;
    MoveL Offs(pOrigin,200.49,317.80,0.00),v40,z0,tPen\WObj:=wPaper;
    MoveL Offs(pOrigin,200.65,316.95,0.00),v40,z0,tPen\WObj:=wPaper;
    MoveL Offs(pOrigin,200.65,315.89,0.00),v40,fine,tPen\WObj:=wPaper;
    MoveL Offs(pOrigin,200.65,315.89,6.00),v60,z5,tPen\WObj:=wPaper;
    MoveL Offs(pOrigin,198.54,315.89,6.00),vTravel,z5,tPen\WObj:=wPaper;
    MoveL Offs(pOrigin,198.54,315.89,0.00),v60,z0,tPen\WObj:=wPaper;
    MoveL Offs(pOrigin,198.54,314.19,0.00),v40,fine,tPen\WObj:=wPaper;
    MoveL Offs(pOrigin,198.54,314.19,6.00),v60,z5,tPen\WObj:=wPaper;
    MoveL Offs(pOrigin,197.73,315.96,6.00),vTravel,z5,tPen\WObj:=wPaper;
    MoveL Offs(pOrigin,197.73,315.96,0.00),v60,z0,tPen\WObj:=wPaper;
    MoveL Offs(pOrigin,203.25,315.96,0.00),v40,z0,tPen\WObj:=wPaper;
    MoveL Offs(pOrigin,203.04,315.67,0.00),v40,z0,tPen\WObj:=wPaper;
    MoveL Offs(pOrigin,203.25,315.25,0.00),v40,z0,tPen\WObj:=wPaper;
    MoveL Offs(pOrigin,203.89,315.04,0.00),v40,z0,tPen\WObj:=wPaper;
    MoveL Offs(pOrigin,203.89,315.04,0.00),v40,z0,tPen\WObj:=wPaper;
    MoveL Offs(pOrigin,204.74,315.04,0.00),v40,z0,tPen\WObj:=wPaper;
    MoveL Offs(pOrigin,205.16,314.40,0.00),v40,z0,tPen\WObj:=wPaper;
    MoveL Offs(pOrigin,204.85,313.62,0.00),v40,z0,tPen\WObj:=wPaper;
    MoveL Offs(pOrigin,197.94,320.53,0.00),v40,fine,tPen\WObj:=wPaper;
    MoveL Offs(pOrigin,197.94,320.53,6.00),v60,z5,tPen\WObj:=wPaper;
    MoveL Offs(pOrigin,197.09,318.65,6.00),vTravel,z5,tPen\WObj:=wPaper;
    MoveL Offs(pOrigin,197.09,318.65,0.00),v60,z0,tPen\WObj:=wPaper;
    MoveL Offs(pOrigin,197.51,319.08,0.00),v40,z0,tPen\WObj:=wPaper;
    MoveL Offs(pOrigin,197.09,318.65,0.00),v40,fine,tPen\WObj:=wPaper;
    MoveL Offs(pOrigin,197.09,318.65,6.00),v60,z5,tPen\WObj:=wPaper;
    MoveL Offs(pOrigin,197.73,317.59,6.00),vTravel,z5,tPen\WObj:=wPaper;
    MoveL Offs(pOrigin,197.73,317.59,0.00),v60,z0,tPen\WObj:=wPaper;
    MoveL Offs(pOrigin,198.15,318.01,0.00),v40,z0,tPen\WObj:=wPaper;
    MoveL Offs(pOrigin,197.73,317.59,0.00),v40,z0,tPen\WObj:=wPaper;
    MoveL Offs(pOrigin,198.36,318.23,0.00),v40,z0,tPen\WObj:=wPaper;
    MoveL Offs(pOrigin,199.21,318.86,0.00),v40,z0,tPen\WObj:=wPaper;
    MoveL Offs(pOrigin,198.36,318.23,0.00),v40,fine,tPen\WObj:=wPaper;
    MoveL Offs(pOrigin,198.36,318.23,6.00),v60,z5,tPen\WObj:=wPaper;
    MoveL Offs(pOrigin,197.94,316.10,6.00),vTravel,z5,tPen\WObj:=wPaper;
    MoveL Offs(pOrigin,197.94,316.10,0.00),v60,z0,tPen\WObj:=wPaper;
    MoveL Offs(pOrigin,198.79,316.95,0.00),v40,z0,tPen\WObj:=wPaper;
    MoveL Offs(pOrigin,197.94,316.10,0.00),v40,fine,tPen\WObj:=wPaper;
    MoveL Offs(pOrigin,197.94,316.10,6.00),v60,z5,tPen\WObj:=wPaper;
    MoveL Offs(pOrigin,195.25,315.74,6.00),vTravel,z5,tPen\WObj:=wPaper;
    MoveL Offs(pOrigin,195.25,315.74,0.00),v60,z0,tPen\WObj:=wPaper;
    MoveL Offs(pOrigin,200.66,310.33,0.00),v40,z0,tPen\WObj:=wPaper;
    MoveL Offs(pOrigin,201.34,309.94,0.00),v40,z0,tPen\WObj:=wPaper;
    MoveL Offs(pOrigin,201.98,310.58,0.00),v40,z0,tPen\WObj:=wPaper;
    MoveL Offs(pOrigin,203.68,310.36,0.00),v40,z0,tPen\WObj:=wPaper;
    MoveL Offs(pOrigin,203.44,311.26,0.00),v40,z0,tPen\WObj:=wPaper;
    MoveL Offs(pOrigin,204.19,312.01,0.00),v40,z0,tPen\WObj:=wPaper;
    MoveL Offs(pOrigin,204.25,312.72,0.00),v40,z0,tPen\WObj:=wPaper;
    MoveL Offs(pOrigin,213.57,303.40,0.00),v40,z0,tPen\WObj:=wPaper;
    MoveL Offs(pOrigin,213.01,304.40,0.00),v40,z0,tPen\WObj:=wPaper;
    MoveL Offs(pOrigin,191.07,282.46,0.00),v40,z0,tPen\WObj:=wPaper;
    MoveL Offs(pOrigin,191.78,282.17,0.00),v40,z0,tPen\WObj:=wPaper;
    MoveL Offs(pOrigin,199.85,282.17,0.00),v40,z0,tPen\WObj:=wPaper;
    MoveL Offs(pOrigin,200.27,281.67,0.00),v40,z0,tPen\WObj:=wPaper;
    MoveL Offs(pOrigin,199.99,280.61,0.00),v40,z0,tPen\WObj:=wPaper;
    MoveL Offs(pOrigin,198.79,279.12,0.00),v40,z0,tPen\WObj:=wPaper;
    MoveL Offs(pOrigin,196.45,278.06,0.00),v40,fine,tPen\WObj:=wPaper;
    MoveL Offs(pOrigin,196.45,278.06,6.00),v60,z5,tPen\WObj:=wPaper;
    MoveL Offs(pOrigin,197.49,277.21,6.00),vTravel,z5,tPen\WObj:=wPaper;
    MoveL Offs(pOrigin,197.49,277.21,0.00),v60,z0,tPen\WObj:=wPaper;
    MoveL Offs(pOrigin,197.49,270.62,0.00),v40,z0,tPen\WObj:=wPaper;
    MoveL Offs(pOrigin,197.09,270.55,0.00),v40,z0,tPen\WObj:=wPaper;
    MoveL Offs(pOrigin,205.59,270.55,0.00),v40,z0,tPen\WObj:=wPaper;
    MoveL Offs(pOrigin,206.17,270.67,0.00),v40,z0,tPen\WObj:=wPaper;
    MoveL Offs(pOrigin,194.90,259.41,0.00),v40,z0,tPen\WObj:=wPaper;
    MoveL Offs(pOrigin,194.53,259.72,0.00),v40,z0,tPen\WObj:=wPaper;
    MoveL Offs(pOrigin,199.03,255.21,0.00),v40,fine,tPen\WObj:=wPaper;
    MoveL Offs(pOrigin,199.03,255.21,6.00),v60,z5,tPen\WObj:=wPaper;
    MoveL Offs(pOrigin,199.04,253.71,6.00),vTravel,z5,tPen\WObj:=wPaper;
    MoveL Offs(pOrigin,199.04,253.71,0.00),v60,z0,tPen\WObj:=wPaper;
    MoveL Offs(pOrigin,194.23,258.52,0.00),v40,z0,tPen\WObj:=wPaper;
    MoveL Offs(pOrigin,194.59,257.61,0.00),v40,z0,tPen\WObj:=wPaper;
    MoveL Offs(pOrigin,196.84,259.86,0.00),v40,fine,tPen\WObj:=wPaper;
    MoveL Offs(pOrigin,196.84,259.86,6.00),v60,z5,tPen\WObj:=wPaper;
    MoveL Offs(pOrigin,197.30,261.70,6.00),vTravel,z5,tPen\WObj:=wPaper;
    MoveL Offs(pOrigin,197.30,261.70,0.00),v60,z0,tPen\WObj:=wPaper;
    MoveL Offs(pOrigin,197.51,262.12,0.00),v40,z0,tPen\WObj:=wPaper;
    MoveL Offs(pOrigin,197.30,261.70,0.00),v40,fine,tPen\WObj:=wPaper;
    MoveL Offs(pOrigin,197.30,261.70,6.00),v60,z5,tPen\WObj:=wPaper;
    MoveL Offs(pOrigin,198.15,262.76,6.00),vTravel,z5,tPen\WObj:=wPaper;
    MoveL Offs(pOrigin,198.15,262.76,0.00),v60,z0,tPen\WObj:=wPaper;
    MoveL Offs(pOrigin,198.57,262.98,0.00),v40,z0,tPen\WObj:=wPaper;
    MoveL Offs(pOrigin,198.15,262.76,0.00),v40,fine,tPen\WObj:=wPaper;
    MoveL Offs(pOrigin,198.15,262.76,6.00),v60,z5,tPen\WObj:=wPaper;
  ENDPROC

  PROC DrawPart183()
    MoveL Offs(pOrigin,197.30,263.83,6.00),vTravel,z5,tPen\WObj:=wPaper;
    MoveL Offs(pOrigin,197.30,263.83,0.00),v60,z0,tPen\WObj:=wPaper;
    MoveL Offs(pOrigin,197.94,264.25,0.00),v40,z0,tPen\WObj:=wPaper;
    MoveL Offs(pOrigin,197.30,263.83,0.00),v40,z0,tPen\WObj:=wPaper;
    MoveL Offs(pOrigin,197.36,264.35,0.00),v40,z0,tPen\WObj:=wPaper;
    MoveL Offs(pOrigin,199.46,262.25,0.00),v40,fine,tPen\WObj:=wPaper;
    MoveL Offs(pOrigin,199.46,262.25,6.00),v60,z5,tPen\WObj:=wPaper;
    MoveL Offs(pOrigin,200.66,261.05,6.00),vTravel,z5,tPen\WObj:=wPaper;
    MoveL Offs(pOrigin,200.66,261.05,0.00),v60,z0,tPen\WObj:=wPaper;
    MoveL Offs(pOrigin,212.84,248.88,0.00),v40,fine,tPen\WObj:=wPaper;
    MoveL Offs(pOrigin,212.84,248.88,6.00),v60,z5,tPen\WObj:=wPaper;
    MoveL Offs(pOrigin,214.78,248.42,6.00),vTravel,z5,tPen\WObj:=wPaper;
    MoveL Offs(pOrigin,214.78,248.42,0.00),v60,z0,tPen\WObj:=wPaper;
    MoveL Offs(pOrigin,198.11,265.10,0.00),v40,fine,tPen\WObj:=wPaper;
    MoveL Offs(pOrigin,198.11,265.10,6.00),v60,z5,tPen\WObj:=wPaper;
    MoveL Offs(pOrigin,199.00,266.33,6.00),vTravel,z5,tPen\WObj:=wPaper;
    MoveL Offs(pOrigin,199.00,266.33,0.00),v60,z0,tPen\WObj:=wPaper;
    MoveL Offs(pOrigin,206.44,266.33,0.00),v40,fine,tPen\WObj:=wPaper;
    MoveL Offs(pOrigin,206.44,266.33,6.00),v60,z5,tPen\WObj:=wPaper;
    MoveL Offs(pOrigin,207.08,268.07,6.00),vTravel,z5,tPen\WObj:=wPaper;
    MoveL Offs(pOrigin,207.08,268.07,0.00),v60,z0,tPen\WObj:=wPaper;
    MoveL Offs(pOrigin,190.10,285.05,0.00),v40,z0,tPen\WObj:=wPaper;
    MoveL Offs(pOrigin,190.63,285.01,0.00),v40,z0,tPen\WObj:=wPaper;
    MoveL Offs(pOrigin,197.24,291.62,0.00),v40,fine,tPen\WObj:=wPaper;
    MoveL Offs(pOrigin,197.24,291.62,6.00),v60,z5,tPen\WObj:=wPaper;
    MoveL Offs(pOrigin,197.94,290.39,6.00),vTravel,z5,tPen\WObj:=wPaper;
    MoveL Offs(pOrigin,197.94,290.39,0.00),v60,z0,tPen\WObj:=wPaper;
    MoveL Offs(pOrigin,198.15,290.81,0.00),v40,z0,tPen\WObj:=wPaper;
    MoveL Offs(pOrigin,197.94,290.39,0.00),v40,fine,tPen\WObj:=wPaper;
    MoveL Offs(pOrigin,197.94,290.39,6.00),v60,z5,tPen\WObj:=wPaper;
    MoveL Offs(pOrigin,198.57,288.90,6.00),vTravel,z5,tPen\WObj:=wPaper;
    MoveL Offs(pOrigin,198.57,288.90,0.00),v60,z0,tPen\WObj:=wPaper;
    MoveL Offs(pOrigin,198.79,289.33,0.00),v40,z0,tPen\WObj:=wPaper;
    MoveL Offs(pOrigin,198.57,288.90,0.00),v40,fine,tPen\WObj:=wPaper;
    MoveL Offs(pOrigin,198.57,288.90,6.00),v60,z5,tPen\WObj:=wPaper;
    MoveL Offs(pOrigin,200.27,289.54,6.00),vTravel,z5,tPen\WObj:=wPaper;
    MoveL Offs(pOrigin,200.27,289.54,0.00),v60,z0,tPen\WObj:=wPaper;
    MoveL Offs(pOrigin,200.49,289.96,0.00),v40,z0,tPen\WObj:=wPaper;
    MoveL Offs(pOrigin,200.27,289.54,0.00),v40,fine,tPen\WObj:=wPaper;
    MoveL Offs(pOrigin,200.27,289.54,6.00),v60,z5,tPen\WObj:=wPaper;
    MoveL Offs(pOrigin,199.43,291.45,6.00),vTravel,z5,tPen\WObj:=wPaper;
    MoveL Offs(pOrigin,199.43,291.45,0.00),v60,z0,tPen\WObj:=wPaper;
    MoveL Offs(pOrigin,200.20,291.88,0.00),v40,z0,tPen\WObj:=wPaper;
    MoveL Offs(pOrigin,201.05,293.15,0.00),v40,z0,tPen\WObj:=wPaper;
    MoveL Offs(pOrigin,201.12,293.79,0.00),v40,z0,tPen\WObj:=wPaper;
    MoveL Offs(pOrigin,200.70,293.78,0.00),v40,z0,tPen\WObj:=wPaper;
    MoveL Offs(pOrigin,205.59,293.78,0.00),v40,z0,tPen\WObj:=wPaper;
    MoveL Offs(pOrigin,204.88,294.42,0.00),v40,z0,tPen\WObj:=wPaper;
    MoveL Offs(pOrigin,204.88,299.10,0.00),v40,fine,tPen\WObj:=wPaper;
    MoveL Offs(pOrigin,204.88,299.10,6.00),v60,z5,tPen\WObj:=wPaper;
    MoveL Offs(pOrigin,203.25,299.06,6.00),vTravel,z5,tPen\WObj:=wPaper;
    MoveL Offs(pOrigin,203.25,299.06,0.00),v60,z0,tPen\WObj:=wPaper;
    MoveL Offs(pOrigin,208.35,299.06,0.00),v40,z0,tPen\WObj:=wPaper;
    MoveL Offs(pOrigin,208.95,298.85,0.00),v40,z0,tPen\WObj:=wPaper;
    MoveL Offs(pOrigin,191.52,281.42,0.00),v40,z0,tPen\WObj:=wPaper;
    MoveL Offs(pOrigin,191.99,281.11,0.00),v40,z0,tPen\WObj:=wPaper;
    MoveL Offs(pOrigin,198.79,281.11,0.00),v40,z0,tPen\WObj:=wPaper;
    MoveL Offs(pOrigin,198.57,280.61,0.00),v40,z0,tPen\WObj:=wPaper;
    MoveL Offs(pOrigin,197.30,279.34,0.00),v40,z0,tPen\WObj:=wPaper;
    MoveL Offs(pOrigin,197.30,279.34,0.00),v40,z0,tPen\WObj:=wPaper;
    MoveL Offs(pOrigin,196.45,279.76,0.00),v40,z0,tPen\WObj:=wPaper;
    MoveL Offs(pOrigin,195.18,278.91,0.00),v40,z0,tPen\WObj:=wPaper;
    MoveL Offs(pOrigin,194.54,278.98,0.00),v40,z0,tPen\WObj:=wPaper;
    MoveL Offs(pOrigin,194.32,279.34,0.00),v40,fine,tPen\WObj:=wPaper;
    MoveL Offs(pOrigin,194.32,279.34,6.00),v60,z5,tPen\WObj:=wPaper;
    MoveL Offs(pOrigin,193.26,278.70,6.00),vTravel,z5,tPen\WObj:=wPaper;
    MoveL Offs(pOrigin,193.26,278.70,0.00),v60,z0,tPen\WObj:=wPaper;
    MoveL Offs(pOrigin,193.26,282.74,0.00),v40,z0,tPen\WObj:=wPaper;
    MoveL Offs(pOrigin,192.84,282.52,0.00),v40,z0,tPen\WObj:=wPaper;
    MoveL Offs(pOrigin,192.98,284.01,0.00),v40,z0,tPen\WObj:=wPaper;
    MoveL Offs(pOrigin,193.90,285.50,0.00),v40,z0,tPen\WObj:=wPaper;
    MoveL Offs(pOrigin,193.69,286.14,0.00),v40,z0,tPen\WObj:=wPaper;
    MoveL Offs(pOrigin,193.69,286.14,0.00),v40,z0,tPen\WObj:=wPaper;
    MoveL Offs(pOrigin,193.90,287.20,0.00),v40,z0,tPen\WObj:=wPaper;
    MoveL Offs(pOrigin,193.90,287.20,0.00),v40,z0,tPen\WObj:=wPaper;
    MoveL Offs(pOrigin,193.26,287.84,0.00),v40,z0,tPen\WObj:=wPaper;
    MoveL Offs(pOrigin,193.69,289.11,0.00),v40,z0,tPen\WObj:=wPaper;
    MoveL Offs(pOrigin,194.32,289.89,0.00),v40,z0,tPen\WObj:=wPaper;
    MoveL Offs(pOrigin,195.10,290.25,0.00),v40,z0,tPen\WObj:=wPaper;
    MoveL Offs(pOrigin,199.21,295.91,0.00),v40,z0,tPen\WObj:=wPaper;
    MoveL Offs(pOrigin,200.91,297.47,0.00),v40,z0,tPen\WObj:=wPaper;
    MoveL Offs(pOrigin,201.98,297.61,0.00),v40,fine,tPen\WObj:=wPaper;
    MoveL Offs(pOrigin,201.98,297.61,6.00),v60,z5,tPen\WObj:=wPaper;
    MoveL Offs(pOrigin,201.34,295.90,6.00),vTravel,z5,tPen\WObj:=wPaper;
    MoveL Offs(pOrigin,201.34,295.90,0.00),v60,z0,tPen\WObj:=wPaper;
    MoveL Offs(pOrigin,206.86,295.90,0.00),v40,z0,tPen\WObj:=wPaper;
    MoveL Offs(pOrigin,205.93,295.70,0.00),v40,z0,tPen\WObj:=wPaper;
    MoveL Offs(pOrigin,205.93,305.47,0.00),v40,fine,tPen\WObj:=wPaper;
    MoveL Offs(pOrigin,205.93,305.47,6.00),v60,z5,tPen\WObj:=wPaper;
    MoveL Offs(pOrigin,206.86,303.77,6.00),vTravel,z5,tPen\WObj:=wPaper;
    MoveL Offs(pOrigin,206.86,303.77,0.00),v60,z0,tPen\WObj:=wPaper;
    MoveL Offs(pOrigin,206.01,303.99,0.00),v40,z0,tPen\WObj:=wPaper;
    MoveL Offs(pOrigin,205.38,303.00,0.00),v40,z0,tPen\WObj:=wPaper;
    MoveL Offs(pOrigin,201.34,301.86,0.00),v40,z0,tPen\WObj:=wPaper;
    MoveL Offs(pOrigin,200.72,301.07,0.00),v40,z0,tPen\WObj:=wPaper;
    MoveL Offs(pOrigin,223.86,324.21,0.00),v40,fine,tPen\WObj:=wPaper;
    MoveL Offs(pOrigin,223.86,324.21,6.00),v60,z5,tPen\WObj:=wPaper;
    MoveL Offs(pOrigin,224.07,322.48,6.00),vTravel,z5,tPen\WObj:=wPaper;
    MoveL Offs(pOrigin,224.07,322.48,0.00),v60,z0,tPen\WObj:=wPaper;
    MoveL Offs(pOrigin,223.37,326.09,0.00),v40,z0,tPen\WObj:=wPaper;
    MoveL Offs(pOrigin,221.95,327.65,0.00),v40,z0,tPen\WObj:=wPaper;
    MoveL Offs(pOrigin,217.91,329.27,0.00),v40,z0,tPen\WObj:=wPaper;
    MoveL Offs(pOrigin,215.57,329.49,0.00),v40,z0,tPen\WObj:=wPaper;
    MoveL Offs(pOrigin,213.45,329.27,0.00),v40,z0,tPen\WObj:=wPaper;
    MoveL Offs(pOrigin,212.60,329.91,0.00),v40,fine,tPen\WObj:=wPaper;
    MoveL Offs(pOrigin,212.60,329.91,6.00),v60,z5,tPen\WObj:=wPaper;
    MoveL Offs(pOrigin,212.27,328.64,6.00),vTravel,z5,tPen\WObj:=wPaper;
    MoveL Offs(pOrigin,212.27,328.64,0.00),v60,z0,tPen\WObj:=wPaper;
    MoveL Offs(pOrigin,212.27,327.58,0.00),v40,fine,tPen\WObj:=wPaper;
    MoveL Offs(pOrigin,212.27,327.58,6.00),v60,z5,tPen\WObj:=wPaper;
    MoveL Offs(pOrigin,210.16,328.00,6.00),vTravel,z5,tPen\WObj:=wPaper;
    MoveL Offs(pOrigin,210.16,328.00,0.00),v60,z0,tPen\WObj:=wPaper;
    MoveL Offs(pOrigin,210.16,326.94,0.00),v40,z0,tPen\WObj:=wPaper;
    MoveL Offs(pOrigin,210.68,325.96,0.00),v40,z0,tPen\WObj:=wPaper;
    MoveL Offs(pOrigin,214.44,329.72,0.00),v40,fine,tPen\WObj:=wPaper;
    MoveL Offs(pOrigin,214.44,329.72,6.00),v60,z5,tPen\WObj:=wPaper;
    MoveL Offs(pOrigin,215.79,331.07,6.00),vTravel,z5,tPen\WObj:=wPaper;
    MoveL Offs(pOrigin,215.79,331.07,0.00),v60,z0,tPen\WObj:=wPaper;
    MoveL Offs(pOrigin,222.85,338.14,0.00),v40,z0,tPen\WObj:=wPaper;
    MoveL Offs(pOrigin,223.35,338.43,0.00),v40,z0,tPen\WObj:=wPaper;
  ENDPROC

  PROC DrawPart184()
    MoveL Offs(pOrigin,234.31,327.46,0.00),v40,fine,tPen\WObj:=wPaper;
    MoveL Offs(pOrigin,234.31,327.46,6.00),v60,z5,tPen\WObj:=wPaper;
    MoveL Offs(pOrigin,234.32,325.96,6.00),vTravel,z5,tPen\WObj:=wPaper;
    MoveL Offs(pOrigin,234.32,325.96,0.00),v60,z0,tPen\WObj:=wPaper;
    MoveL Offs(pOrigin,232.52,327.76,0.00),v40,z0,tPen\WObj:=wPaper;
    MoveL Offs(pOrigin,231.47,327.32,0.00),v40,z0,tPen\WObj:=wPaper;
    MoveL Offs(pOrigin,221.10,337.68,0.00),v40,z0,tPen\WObj:=wPaper;
    MoveL Offs(pOrigin,220.30,337.08,0.00),v40,z0,tPen\WObj:=wPaper;
    MoveL Offs(pOrigin,193.10,309.88,0.00),v40,z0,tPen\WObj:=wPaper;
    MoveL Offs(pOrigin,193.17,310.36,0.00),v40,z0,tPen\WObj:=wPaper;
    MoveL Offs(pOrigin,198.58,304.95,0.00),v40,z0,tPen\WObj:=wPaper;
    MoveL Offs(pOrigin,198.57,305.48,0.00),v40,z0,tPen\WObj:=wPaper;
    MoveL Offs(pOrigin,199.00,305.90,0.00),v40,z0,tPen\WObj:=wPaper;
    MoveL Offs(pOrigin,198.57,305.48,0.00),v40,z0,tPen\WObj:=wPaper;
    MoveL Offs(pOrigin,197.51,305.40,0.00),v40,z0,tPen\WObj:=wPaper;
    MoveL Offs(pOrigin,195.81,305.40,0.00),v40,z0,tPen\WObj:=wPaper;
    MoveL Offs(pOrigin,195.19,305.99,0.00),v40,z0,tPen\WObj:=wPaper;
    MoveL Offs(pOrigin,190.38,301.19,0.00),v40,z0,tPen\WObj:=wPaper;
    MoveL Offs(pOrigin,189.90,301.68,0.00),v40,z0,tPen\WObj:=wPaper;
    MoveL Offs(pOrigin,205.53,286.05,0.00),v40,z0,tPen\WObj:=wPaper;
    MoveL Offs(pOrigin,204.86,285.80,0.00),v40,z0,tPen\WObj:=wPaper;
    MoveL Offs(pOrigin,194.04,274.98,0.00),v40,z0,tPen\WObj:=wPaper;
    MoveL Offs(pOrigin,194.32,274.45,0.00),v40,z0,tPen\WObj:=wPaper;
    MoveL Offs(pOrigin,193.48,275.51,0.00),v40,z0,tPen\WObj:=wPaper;
    MoveL Offs(pOrigin,194.32,274.45,0.00),v40,fine,tPen\WObj:=wPaper;
    MoveL Offs(pOrigin,194.32,274.45,6.00),v60,z5,tPen\WObj:=wPaper;
    MoveL Offs(pOrigin,195.39,273.72,6.00),vTravel,z5,tPen\WObj:=wPaper;
    MoveL Offs(pOrigin,195.39,273.72,0.00),v60,z0,tPen\WObj:=wPaper;
    MoveL Offs(pOrigin,204.95,273.72,0.00),v40,z0,tPen\WObj:=wPaper;
    MoveL Offs(pOrigin,205.28,274.27,0.00),v40,z0,tPen\WObj:=wPaper;
    MoveL Offs(pOrigin,198.22,267.20,0.00),v40,z0,tPen\WObj:=wPaper;
    MoveL Offs(pOrigin,198.57,266.59,0.00),v40,z0,tPen\WObj:=wPaper;
    MoveL Offs(pOrigin,198.15,267.01,0.00),v40,z0,tPen\WObj:=wPaper;
    MoveL Offs(pOrigin,198.57,266.59,0.00),v40,fine,tPen\WObj:=wPaper;
    MoveL Offs(pOrigin,198.57,266.59,6.00),v60,z5,tPen\WObj:=wPaper;
    MoveL Offs(pOrigin,197.35,267.35,6.00),vTravel,z5,tPen\WObj:=wPaper;
    MoveL Offs(pOrigin,197.35,267.35,0.00),v60,z0,tPen\WObj:=wPaper;
    MoveL Offs(pOrigin,209.82,254.88,0.00),v40,fine,tPen\WObj:=wPaper;
    MoveL Offs(pOrigin,209.82,254.88,6.00),v60,z5,tPen\WObj:=wPaper;
    MoveL Offs(pOrigin,208.51,255.10,6.00),vTravel,z5,tPen\WObj:=wPaper;
    MoveL Offs(pOrigin,208.51,255.10,0.00),v60,z0,tPen\WObj:=wPaper;
    MoveL Offs(pOrigin,204.46,251.05,0.00),v40,z0,tPen\WObj:=wPaper;
    MoveL Offs(pOrigin,204.95,251.54,0.00),v40,z0,tPen\WObj:=wPaper;
    MoveL Offs(pOrigin,206.86,251.54,0.00),v40,z0,tPen\WObj:=wPaper;
    MoveL Offs(pOrigin,207.45,251.05,0.00),v40,z0,tPen\WObj:=wPaper;
    MoveL Offs(pOrigin,205.05,248.65,0.00),v40,z0,tPen\WObj:=wPaper;
    MoveL Offs(pOrigin,204.45,248.30,0.00),v40,z0,tPen\WObj:=wPaper;
    MoveL Offs(pOrigin,207.45,245.30,0.00),v40,fine,tPen\WObj:=wPaper;
    MoveL Offs(pOrigin,207.45,245.30,6.00),v60,z5,tPen\WObj:=wPaper;
    MoveL Offs(pOrigin,206.68,244.31,6.00),vTravel,z5,tPen\WObj:=wPaper;
    MoveL Offs(pOrigin,206.68,244.31,0.00),v60,z0,tPen\WObj:=wPaper;
    MoveL Offs(pOrigin,204.88,242.51,0.00),v40,z0,tPen\WObj:=wPaper;
    MoveL Offs(pOrigin,205.48,241.61,0.00),v40,z0,tPen\WObj:=wPaper;
    MoveL Offs(pOrigin,206.98,243.11,0.00),v40,z0,tPen\WObj:=wPaper;
    MoveL Offs(pOrigin,207.46,243.80,0.00),v40,z0,tPen\WObj:=wPaper;
    MoveL Offs(pOrigin,204.30,246.96,0.00),v40,z0,tPen\WObj:=wPaper;
    MoveL Offs(pOrigin,203.86,245.91,0.00),v40,z0,tPen\WObj:=wPaper;
    MoveL Offs(pOrigin,207.46,242.30,0.00),v40,fine,tPen\WObj:=wPaper;
    MoveL Offs(pOrigin,207.46,242.30,6.00),v60,z5,tPen\WObj:=wPaper;
    MoveL Offs(pOrigin,207.17,239.61,6.00),vTravel,z5,tPen\WObj:=wPaper;
    MoveL Offs(pOrigin,207.17,239.61,0.00),v60,z0,tPen\WObj:=wPaper;
    MoveL Offs(pOrigin,194.70,252.08,0.00),v40,z0,tPen\WObj:=wPaper;
    MoveL Offs(pOrigin,195.17,252.22,0.00),v40,z0,tPen\WObj:=wPaper;
    MoveL Offs(pOrigin,196.53,253.57,0.00),v40,z0,tPen\WObj:=wPaper;
    MoveL Offs(pOrigin,196.97,252.52,0.00),v40,z0,tPen\WObj:=wPaper;
    MoveL Offs(pOrigin,195.62,251.17,0.00),v40,fine,tPen\WObj:=wPaper;
    MoveL Offs(pOrigin,195.62,251.17,6.00),v60,z5,tPen\WObj:=wPaper;
    MoveL Offs(pOrigin,194.88,253.41,6.00),vTravel,z5,tPen\WObj:=wPaper;
    MoveL Offs(pOrigin,194.88,253.41,0.00),v60,z0,tPen\WObj:=wPaper;
    MoveL Offs(pOrigin,196.38,254.92,0.00),v40,fine,tPen\WObj:=wPaper;
    MoveL Offs(pOrigin,196.38,254.92,6.00),v60,z5,tPen\WObj:=wPaper;
    MoveL Offs(pOrigin,194.24,257.02,6.00),vTravel,z5,tPen\WObj:=wPaper;
    MoveL Offs(pOrigin,194.24,257.02,0.00),v60,z0,tPen\WObj:=wPaper;
    MoveL Offs(pOrigin,202.35,248.91,0.00),v40,fine,tPen\WObj:=wPaper;
    MoveL Offs(pOrigin,202.35,248.91,6.00),v60,z5,tPen\WObj:=wPaper;
    MoveL Offs(pOrigin,201.12,249.59,6.00),vTravel,z5,tPen\WObj:=wPaper;
    MoveL Offs(pOrigin,201.12,249.59,0.00),v60,z0,tPen\WObj:=wPaper;
    MoveL Offs(pOrigin,201.55,256.81,0.00),v40,z0,tPen\WObj:=wPaper;
    MoveL Offs(pOrigin,202.33,256.40,0.00),v40,z0,tPen\WObj:=wPaper;
    MoveL Offs(pOrigin,207.89,250.84,0.00),v40,z0,tPen\WObj:=wPaper;
    MoveL Offs(pOrigin,206.86,250.49,0.00),v40,z0,tPen\WObj:=wPaper;
    MoveL Offs(pOrigin,205.38,250.49,0.00),v40,fine,tPen\WObj:=wPaper;
    MoveL Offs(pOrigin,205.38,250.49,6.00),v60,z5,tPen\WObj:=wPaper;
    MoveL Offs(pOrigin,203.54,252.20,6.00),vTravel,z5,tPen\WObj:=wPaper;
    MoveL Offs(pOrigin,203.54,252.20,0.00),v60,z0,tPen\WObj:=wPaper;
    MoveL Offs(pOrigin,207.74,247.99,0.00),v40,fine,tPen\WObj:=wPaper;
    MoveL Offs(pOrigin,207.74,247.99,6.00),v60,z5,tPen\WObj:=wPaper;
    MoveL Offs(pOrigin,207.89,249.34,6.00),vTravel,z5,tPen\WObj:=wPaper;
    MoveL Offs(pOrigin,207.89,249.34,0.00),v60,z0,tPen\WObj:=wPaper;
    MoveL Offs(pOrigin,202.78,254.45,0.00),v40,fine,tPen\WObj:=wPaper;
    MoveL Offs(pOrigin,202.78,254.45,6.00),v60,z5,tPen\WObj:=wPaper;
    MoveL Offs(pOrigin,203.87,253.44,6.00),vTravel,z5,tPen\WObj:=wPaper;
    MoveL Offs(pOrigin,203.87,253.44,0.00),v60,z0,tPen\WObj:=wPaper;
    MoveL Offs(pOrigin,208.22,257.80,0.00),v40,z0,tPen\WObj:=wPaper;
    MoveL Offs(pOrigin,207.71,257.66,0.00),v40,z0,tPen\WObj:=wPaper;
    MoveL Offs(pOrigin,208.14,258.09,0.00),v40,z0,tPen\WObj:=wPaper;
    MoveL Offs(pOrigin,207.71,257.66,0.00),v40,fine,tPen\WObj:=wPaper;
    MoveL Offs(pOrigin,207.71,257.66,6.00),v60,z5,tPen\WObj:=wPaper;
    MoveL Offs(pOrigin,208.30,260.88,6.00),vTravel,z5,tPen\WObj:=wPaper;
    MoveL Offs(pOrigin,208.30,260.88,0.00),v60,z0,tPen\WObj:=wPaper;
    MoveL Offs(pOrigin,192.38,276.80,0.00),v40,fine,tPen\WObj:=wPaper;
    MoveL Offs(pOrigin,192.38,276.80,6.00),v60,z5,tPen\WObj:=wPaper;
    MoveL Offs(pOrigin,194.32,275.94,6.00),vTravel,z5,tPen\WObj:=wPaper;
    MoveL Offs(pOrigin,194.32,275.94,0.00),v60,z0,tPen\WObj:=wPaper;
    MoveL Offs(pOrigin,194.32,284.22,0.00),v40,z0,tPen\WObj:=wPaper;
    MoveL Offs(pOrigin,195.37,284.65,0.00),v40,z0,tPen\WObj:=wPaper;
    MoveL Offs(pOrigin,195.37,283.16,0.00),v40,fine,tPen\WObj:=wPaper;
    MoveL Offs(pOrigin,195.37,283.16,6.00),v60,z5,tPen\WObj:=wPaper;
    MoveL Offs(pOrigin,196.66,283.22,6.00),vTravel,z5,tPen\WObj:=wPaper;
    MoveL Offs(pOrigin,196.66,283.22,0.00),v60,z0,tPen\WObj:=wPaper;
    MoveL Offs(pOrigin,191.56,283.22,0.00),v40,z0,tPen\WObj:=wPaper;
    MoveL Offs(pOrigin,190.41,283.25,0.00),v40,z0,tPen\WObj:=wPaper;
    MoveL Offs(pOrigin,209.04,264.62,0.00),v40,z0,tPen\WObj:=wPaper;
    MoveL Offs(pOrigin,208.45,263.72,0.00),v40,z0,tPen\WObj:=wPaper;
    MoveL Offs(pOrigin,190.87,281.30,0.00),v40,fine,tPen\WObj:=wPaper;
    MoveL Offs(pOrigin,190.87,281.30,6.00),v60,z5,tPen\WObj:=wPaper;
    MoveL Offs(pOrigin,191.62,279.05,6.00),vTravel,z5,tPen\WObj:=wPaper;
    MoveL Offs(pOrigin,191.62,279.05,0.00),v60,z0,tPen\WObj:=wPaper;
    MoveL Offs(pOrigin,208.30,262.37,0.00),v40,fine,tPen\WObj:=wPaper;
    MoveL Offs(pOrigin,208.30,262.37,6.00),v60,z5,tPen\WObj:=wPaper;
  ENDPROC

  PROC DrawPart185()
    MoveL Offs(pOrigin,206.14,261.69,6.00),vTravel,z5,tPen\WObj:=wPaper;
    MoveL Offs(pOrigin,206.14,261.69,0.00),v60,z0,tPen\WObj:=wPaper;
    MoveL Offs(pOrigin,202.38,257.93,0.00),v40,z0,tPen\WObj:=wPaper;
    MoveL Offs(pOrigin,201.63,258.68,0.00),v40,z0,tPen\WObj:=wPaper;
    MoveL Offs(pOrigin,205.09,262.13,0.00),v40,fine,tPen\WObj:=wPaper;
    MoveL Offs(pOrigin,205.09,262.13,6.00),v60,z5,tPen\WObj:=wPaper;
    MoveL Offs(pOrigin,204.88,260.64,6.00),vTravel,z5,tPen\WObj:=wPaper;
    MoveL Offs(pOrigin,204.88,260.64,0.00),v60,z0,tPen\WObj:=wPaper;
    MoveL Offs(pOrigin,204.88,252.99,0.00),v40,z0,tPen\WObj:=wPaper;
    MoveL Offs(pOrigin,204.31,253.66,0.00),v40,z0,tPen\WObj:=wPaper;
    MoveL Offs(pOrigin,206.86,253.66,0.00),v40,fine,tPen\WObj:=wPaper;
    MoveL Offs(pOrigin,206.86,253.66,6.00),v60,z5,tPen\WObj:=wPaper;
    MoveL Offs(pOrigin,208.18,252.04,6.00),vTravel,z5,tPen\WObj:=wPaper;
    MoveL Offs(pOrigin,208.18,252.04,0.00),v60,z0,tPen\WObj:=wPaper;
    MoveL Offs(pOrigin,196.61,263.61,0.00),v40,fine,tPen\WObj:=wPaper;
    MoveL Offs(pOrigin,196.61,263.61,6.00),v60,z5,tPen\WObj:=wPaper;
    MoveL Offs(pOrigin,201.71,263.19,6.00),vTravel,z5,tPen\WObj:=wPaper;
    MoveL Offs(pOrigin,201.71,263.19,0.00),v60,z0,tPen\WObj:=wPaper;
    MoveL Offs(pOrigin,201.71,266.59,0.00),v40,fine,tPen\WObj:=wPaper;
    MoveL Offs(pOrigin,201.71,266.59,6.00),v60,z5,tPen\WObj:=wPaper;
    MoveL Offs(pOrigin,206.78,269.87,6.00),vTravel,z5,tPen\WObj:=wPaper;
    MoveL Offs(pOrigin,206.78,269.87,0.00),v60,z0,tPen\WObj:=wPaper;
    MoveL Offs(pOrigin,190.10,286.55,0.00),v40,z0,tPen\WObj:=wPaper;
    MoveL Offs(pOrigin,190.63,286.51,0.00),v40,z0,tPen\WObj:=wPaper;
    MoveL Offs(pOrigin,228.20,324.07,0.00),v40,z0,tPen\WObj:=wPaper;
    MoveL Offs(pOrigin,228.80,323.17,0.00),v40,z0,tPen\WObj:=wPaper;
    MoveL Offs(pOrigin,199.65,294.02,0.00),v40,fine,tPen\WObj:=wPaper;
    MoveL Offs(pOrigin,199.65,294.02,6.00),v60,z5,tPen\WObj:=wPaper;
    MoveL Offs(pOrigin,201.12,294.64,6.00),vTravel,z5,tPen\WObj:=wPaper;
    MoveL Offs(pOrigin,201.12,294.64,0.00),v60,z0,tPen\WObj:=wPaper;
    MoveL Offs(pOrigin,199.64,294.71,0.00),v40,z0,tPen\WObj:=wPaper;
    MoveL Offs(pOrigin,198.36,293.58,0.00),v40,z0,tPen\WObj:=wPaper;
    MoveL Offs(pOrigin,196.17,290.17,0.00),v40,z0,tPen\WObj:=wPaper;
    MoveL Offs(pOrigin,194.96,287.62,0.00),v40,z0,tPen\WObj:=wPaper;
    MoveL Offs(pOrigin,193.90,287.20,0.00),v40,z0,tPen\WObj:=wPaper;
    MoveL Offs(pOrigin,193.48,286.39,0.00),v40,z0,tPen\WObj:=wPaper;
    MoveL Offs(pOrigin,191.14,286.39,0.00),v40,z0,tPen\WObj:=wPaper;
    MoveL Offs(pOrigin,191.14,285.34,0.00),v40,z0,tPen\WObj:=wPaper;
    MoveL Offs(pOrigin,192.84,285.34,0.00),v40,z0,tPen\WObj:=wPaper;
    MoveL Offs(pOrigin,192.21,285.71,0.00),v40,z0,tPen\WObj:=wPaper;
    MoveL Offs(pOrigin,192.21,291.88,0.00),v40,z0,tPen\WObj:=wPaper;
    MoveL Offs(pOrigin,191.78,291.67,0.00),v40,z0,tPen\WObj:=wPaper;
    MoveL Offs(pOrigin,194.32,291.67,0.00),v40,z0,tPen\WObj:=wPaper;
    MoveL Offs(pOrigin,194.54,292.73,0.00),v40,z0,tPen\WObj:=wPaper;
    MoveL Offs(pOrigin,192.41,292.73,0.00),v40,z0,tPen\WObj:=wPaper;
    MoveL Offs(pOrigin,193.26,292.30,0.00),v40,z0,tPen\WObj:=wPaper;
    MoveL Offs(pOrigin,193.26,290.39,0.00),v40,z0,tPen\WObj:=wPaper;
    MoveL Offs(pOrigin,193.90,290.62,0.00),v40,z0,tPen\WObj:=wPaper;
    MoveL Offs(pOrigin,191.78,290.62,0.00),v40,fine,tPen\WObj:=wPaper;
    MoveL Offs(pOrigin,191.78,290.62,6.00),v60,z5,tPen\WObj:=wPaper;
    MoveL Offs(pOrigin,190.54,290.59,6.00),vTravel,z5,tPen\WObj:=wPaper;
    MoveL Offs(pOrigin,190.54,290.59,0.00),v60,z0,tPen\WObj:=wPaper;
    MoveL Offs(pOrigin,205.71,275.41,0.00),v40,fine,tPen\WObj:=wPaper;
    MoveL Offs(pOrigin,205.71,275.41,6.00),v60,z5,tPen\WObj:=wPaper;
    MoveL Offs(pOrigin,205.87,273.77,6.00),vTravel,z5,tPen\WObj:=wPaper;
    MoveL Offs(pOrigin,205.87,273.77,0.00),v60,z0,tPen\WObj:=wPaper;
    MoveL Offs(pOrigin,190.54,289.09,0.00),v40,z0,tPen\WObj:=wPaper;
    MoveL Offs(pOrigin,190.94,288.30,0.00),v40,z0,tPen\WObj:=wPaper;
    MoveL Offs(pOrigin,195.60,292.96,0.00),v40,z0,tPen\WObj:=wPaper;
    MoveL Offs(pOrigin,195.18,292.73,0.00),v40,z0,tPen\WObj:=wPaper;
    MoveL Offs(pOrigin,195.60,293.36,0.00),v40,z0,tPen\WObj:=wPaper;
    MoveL Offs(pOrigin,195.18,292.73,0.00),v40,fine,tPen\WObj:=wPaper;
    MoveL Offs(pOrigin,195.18,292.73,6.00),v60,z5,tPen\WObj:=wPaper;
    MoveL Offs(pOrigin,194.54,293.78,6.00),vTravel,z5,tPen\WObj:=wPaper;
    MoveL Offs(pOrigin,194.54,293.78,0.00),v60,z0,tPen\WObj:=wPaper;
    MoveL Offs(pOrigin,192.62,293.78,0.00),v40,z0,tPen\WObj:=wPaper;
    MoveL Offs(pOrigin,193.26,294.21,0.00),v40,z0,tPen\WObj:=wPaper;
    MoveL Offs(pOrigin,193.26,296.34,0.00),v40,fine,tPen\WObj:=wPaper;
    MoveL Offs(pOrigin,193.26,296.34,6.00),v60,z5,tPen\WObj:=wPaper;
    MoveL Offs(pOrigin,192.41,294.84,6.00),vTravel,z5,tPen\WObj:=wPaper;
    MoveL Offs(pOrigin,192.41,294.84,0.00),v60,z0,tPen\WObj:=wPaper;
    MoveL Offs(pOrigin,194.54,294.84,0.00),v40,z0,tPen\WObj:=wPaper;
    MoveL Offs(pOrigin,194.96,295.06,0.00),v40,z0,tPen\WObj:=wPaper;
    MoveL Offs(pOrigin,195.88,298.67,0.00),v40,z0,tPen\WObj:=wPaper;
    MoveL Offs(pOrigin,198.36,302.29,0.00),v40,fine,tPen\WObj:=wPaper;
    MoveL Offs(pOrigin,198.36,302.29,6.00),v60,z5,tPen\WObj:=wPaper;
    MoveL Offs(pOrigin,198.44,303.60,6.00),vTravel,z5,tPen\WObj:=wPaper;
    MoveL Offs(pOrigin,198.44,303.60,0.00),v60,z0,tPen\WObj:=wPaper;
    MoveL Offs(pOrigin,207.90,294.13,0.00),v40,fine,tPen\WObj:=wPaper;
    MoveL Offs(pOrigin,207.90,294.13,6.00),v60,z5,tPen\WObj:=wPaper;
    MoveL Offs(pOrigin,206.23,294.84,6.00),vTravel,z5,tPen\WObj:=wPaper;
    MoveL Offs(pOrigin,206.23,294.84,0.00),v60,z0,tPen\WObj:=wPaper;
    MoveL Offs(pOrigin,201.34,294.84,0.00),v40,fine,tPen\WObj:=wPaper;
    MoveL Offs(pOrigin,201.34,294.84,6.00),v60,z5,tPen\WObj:=wPaper;
    MoveL Offs(pOrigin,199.43,296.34,6.00),vTravel,z5,tPen\WObj:=wPaper;
    MoveL Offs(pOrigin,199.43,296.34,0.00),v60,z0,tPen\WObj:=wPaper;
    MoveL Offs(pOrigin,200.27,297.19,0.00),v40,z0,tPen\WObj:=wPaper;
    MoveL Offs(pOrigin,199.43,296.34,0.00),v40,z0,tPen\WObj:=wPaper;
    MoveL Offs(pOrigin,198.79,295.49,0.00),v40,z0,tPen\WObj:=wPaper;
    MoveL Offs(pOrigin,199.21,296.12,0.00),v40,z0,tPen\WObj:=wPaper;
    MoveL Offs(pOrigin,198.79,295.49,0.00),v40,fine,tPen\WObj:=wPaper;
    MoveL Offs(pOrigin,198.79,295.49,6.00),v60,z5,tPen\WObj:=wPaper;
    MoveL Offs(pOrigin,197.73,294.42,6.00),vTravel,z5,tPen\WObj:=wPaper;
    MoveL Offs(pOrigin,197.73,294.42,0.00),v60,z0,tPen\WObj:=wPaper;
    MoveL Offs(pOrigin,198.15,294.85,0.00),v40,z0,tPen\WObj:=wPaper;
    MoveL Offs(pOrigin,197.73,294.42,0.00),v40,fine,tPen\WObj:=wPaper;
    MoveL Offs(pOrigin,197.73,294.42,6.00),v60,z5,tPen\WObj:=wPaper;
    MoveL Offs(pOrigin,196.45,295.49,6.00),vTravel,z5,tPen\WObj:=wPaper;
    MoveL Offs(pOrigin,196.45,295.49,0.00),v60,z0,tPen\WObj:=wPaper;
    MoveL Offs(pOrigin,194.96,295.06,0.00),v40,z0,tPen\WObj:=wPaper;
    MoveL Offs(pOrigin,194.96,295.06,0.00),v40,z0,tPen\WObj:=wPaper;
    MoveL Offs(pOrigin,193.26,291.88,0.00),v40,fine,tPen\WObj:=wPaper;
    MoveL Offs(pOrigin,193.26,291.88,6.00),v60,z5,tPen\WObj:=wPaper;
    MoveL Offs(pOrigin,194.11,289.96,6.00),vTravel,z5,tPen\WObj:=wPaper;
    MoveL Offs(pOrigin,194.11,289.96,0.00),v60,z0,tPen\WObj:=wPaper;
    MoveL Offs(pOrigin,196.31,294.42,0.00),v40,z0,tPen\WObj:=wPaper;
    MoveL Offs(pOrigin,196.45,295.49,0.00),v40,fine,tPen\WObj:=wPaper;
    MoveL Offs(pOrigin,196.45,295.49,6.00),v60,z5,tPen\WObj:=wPaper;
    MoveL Offs(pOrigin,193.69,298.01,6.00),vTravel,z5,tPen\WObj:=wPaper;
    MoveL Offs(pOrigin,193.69,298.01,0.00),v60,z0,tPen\WObj:=wPaper;
    MoveL Offs(pOrigin,191.78,298.01,0.00),v40,z0,tPen\WObj:=wPaper;
    MoveL Offs(pOrigin,191.56,299.06,0.00),v40,z0,tPen\WObj:=wPaper;
    MoveL Offs(pOrigin,193.48,299.06,0.00),v40,z0,tPen\WObj:=wPaper;
    MoveL Offs(pOrigin,193.26,300.16,0.00),v40,z0,tPen\WObj:=wPaper;
    MoveL Offs(pOrigin,193.90,303.99,0.00),v40,z0,tPen\WObj:=wPaper;
    MoveL Offs(pOrigin,194.54,304.34,0.00),v40,z0,tPen\WObj:=wPaper;
    MoveL Offs(pOrigin,196.45,304.34,0.00),v40,z0,tPen\WObj:=wPaper;
    MoveL Offs(pOrigin,196.24,303.56,0.00),v40,z0,tPen\WObj:=wPaper;
    MoveL Offs(pOrigin,196.66,303.99,0.00),v40,z0,tPen\WObj:=wPaper;
    MoveL Offs(pOrigin,196.24,303.56,0.00),v40,fine,tPen\WObj:=wPaper;
  ENDPROC

  PROC DrawPart186()
    MoveL Offs(pOrigin,196.24,303.56,6.00),v60,z5,tPen\WObj:=wPaper;
    MoveL Offs(pOrigin,197.69,304.35,6.00),vTravel,z5,tPen\WObj:=wPaper;
    MoveL Offs(pOrigin,197.69,304.35,0.00),v60,z0,tPen\WObj:=wPaper;
    MoveL Offs(pOrigin,192.73,309.31,0.00),v40,fine,tPen\WObj:=wPaper;
    MoveL Offs(pOrigin,192.73,309.31,6.00),v60,z5,tPen\WObj:=wPaper;
    MoveL Offs(pOrigin,193.90,309.62,6.00),vTravel,z5,tPen\WObj:=wPaper;
    MoveL Offs(pOrigin,193.90,309.62,0.00),v60,z0,tPen\WObj:=wPaper;
    MoveL Offs(pOrigin,196.45,309.62,0.00),v40,fine,tPen\WObj:=wPaper;
    MoveL Offs(pOrigin,196.45,309.62,6.00),v60,z5,tPen\WObj:=wPaper;
    MoveL Offs(pOrigin,194.75,307.51,6.00),vTravel,z5,tPen\WObj:=wPaper;
    MoveL Offs(pOrigin,194.75,307.51,0.00),v60,z0,tPen\WObj:=wPaper;
    MoveL Offs(pOrigin,193.05,307.51,0.00),v40,z0,tPen\WObj:=wPaper;
    MoveL Offs(pOrigin,192.84,306.46,0.00),v40,z0,tPen\WObj:=wPaper;
    MoveL Offs(pOrigin,193.90,306.46,0.00),v40,z0,tPen\WObj:=wPaper;
    MoveL Offs(pOrigin,194.11,306.11,0.00),v40,z0,tPen\WObj:=wPaper;
    MoveL Offs(pOrigin,194.54,306.54,0.00),v40,z0,tPen\WObj:=wPaper;
    MoveL Offs(pOrigin,194.11,306.11,0.00),v40,z0,tPen\WObj:=wPaper;
    MoveL Offs(pOrigin,194.75,306.96,0.00),v40,z0,tPen\WObj:=wPaper;
    MoveL Offs(pOrigin,195.60,307.81,0.00),v40,z0,tPen\WObj:=wPaper;
    MoveL Offs(pOrigin,194.75,306.96,0.00),v40,fine,tPen\WObj:=wPaper;
    MoveL Offs(pOrigin,194.75,306.96,6.00),v60,z5,tPen\WObj:=wPaper;
    MoveL Offs(pOrigin,191.98,307.06,6.00),vTravel,z5,tPen\WObj:=wPaper;
    MoveL Offs(pOrigin,191.98,307.06,0.00),v60,z0,tPen\WObj:=wPaper;
    MoveL Offs(pOrigin,198.15,300.90,0.00),v40,z0,tPen\WObj:=wPaper;
    MoveL Offs(pOrigin,197.30,300.38,0.00),v40,z0,tPen\WObj:=wPaper;
    MoveL Offs(pOrigin,197.94,301.23,0.00),v40,z0,tPen\WObj:=wPaper;
    MoveL Offs(pOrigin,197.30,300.38,0.00),v40,z0,tPen\WObj:=wPaper;
    MoveL Offs(pOrigin,197.55,300.01,0.00),v40,z0,tPen\WObj:=wPaper;
    MoveL Offs(pOrigin,191.69,305.87,0.00),v40,fine,tPen\WObj:=wPaper;
    MoveL Offs(pOrigin,191.69,305.87,6.00),v60,z5,tPen\WObj:=wPaper;
    MoveL Offs(pOrigin,190.65,303.92,6.00),vTravel,z5,tPen\WObj:=wPaper;
    MoveL Offs(pOrigin,190.65,303.92,0.00),v60,z0,tPen\WObj:=wPaper;
    MoveL Offs(pOrigin,206.27,288.29,0.00),v40,z0,tPen\WObj:=wPaper;
    MoveL Offs(pOrigin,205.83,287.25,0.00),v40,z0,tPen\WObj:=wPaper;
    MoveL Offs(pOrigin,190.20,302.87,0.00),v40,z0,tPen\WObj:=wPaper;
    MoveL Offs(pOrigin,190.71,303.35,0.00),v40,z0,tPen\WObj:=wPaper;
    MoveL Offs(pOrigin,190.93,303.77,0.00),v40,z0,tPen\WObj:=wPaper;
    MoveL Offs(pOrigin,190.71,303.35,0.00),v40,fine,tPen\WObj:=wPaper;
    MoveL Offs(pOrigin,190.71,303.35,6.00),v60,z5,tPen\WObj:=wPaper;
    MoveL Offs(pOrigin,189.46,300.63,6.00),vTravel,z5,tPen\WObj:=wPaper;
    MoveL Offs(pOrigin,189.46,300.63,0.00),v60,z0,tPen\WObj:=wPaper;
    MoveL Offs(pOrigin,205.39,284.70,0.00),v40,fine,tPen\WObj:=wPaper;
    MoveL Offs(pOrigin,205.39,284.70,6.00),v60,z5,tPen\WObj:=wPaper;
    MoveL Offs(pOrigin,204.31,285.34,6.00),vTravel,z5,tPen\WObj:=wPaper;
    MoveL Offs(pOrigin,204.31,285.34,0.00),v60,z0,tPen\WObj:=wPaper;
    MoveL Offs(pOrigin,195.18,285.34,0.00),v40,z0,tPen\WObj:=wPaper;
    MoveL Offs(pOrigin,194.96,285.50,0.00),v40,z0,tPen\WObj:=wPaper;
    MoveL Offs(pOrigin,195.18,285.92,0.00),v40,z0,tPen\WObj:=wPaper;
    MoveL Offs(pOrigin,194.96,285.50,0.00),v40,fine,tPen\WObj:=wPaper;
    MoveL Offs(pOrigin,194.96,285.50,6.00),v60,z5,tPen\WObj:=wPaper;
    MoveL Offs(pOrigin,193.69,286.14,6.00),vTravel,z5,tPen\WObj:=wPaper;
    MoveL Offs(pOrigin,193.69,286.14,0.00),v60,z0,tPen\WObj:=wPaper;
    MoveL Offs(pOrigin,192.84,285.29,0.00),v40,z0,tPen\WObj:=wPaper;
    MoveL Offs(pOrigin,193.05,284.44,0.00),v40,fine,tPen\WObj:=wPaper;
    MoveL Offs(pOrigin,193.05,284.44,6.00),v60,z5,tPen\WObj:=wPaper;
    MoveL Offs(pOrigin,193.48,288.50,6.00),vTravel,z5,tPen\WObj:=wPaper;
    MoveL Offs(pOrigin,193.48,288.50,0.00),v60,z0,tPen\WObj:=wPaper;
    MoveL Offs(pOrigin,191.35,288.50,0.00),v40,fine,tPen\WObj:=wPaper;
    MoveL Offs(pOrigin,191.35,288.50,6.00),v60,z5,tPen\WObj:=wPaper;
    MoveL Offs(pOrigin,195.81,291.66,6.00),vTravel,z5,tPen\WObj:=wPaper;
    MoveL Offs(pOrigin,195.81,291.66,0.00),v60,z0,tPen\WObj:=wPaper;
    MoveL Offs(pOrigin,196.24,292.30,0.00),v40,z0,tPen\WObj:=wPaper;
    MoveL Offs(pOrigin,195.81,291.66,0.00),v40,fine,tPen\WObj:=wPaper;
    MoveL Offs(pOrigin,195.81,291.66,6.00),v60,z5,tPen\WObj:=wPaper;
    MoveL Offs(pOrigin,189.02,296.59,6.00),vTravel,z5,tPen\WObj:=wPaper;
    MoveL Offs(pOrigin,189.02,296.59,0.00),v60,z0,tPen\WObj:=wPaper;
    MoveL Offs(pOrigin,205.25,280.36,0.00),v40,z0,tPen\WObj:=wPaper;
    MoveL Offs(pOrigin,204.55,281.01,0.00),v40,z0,tPen\WObj:=wPaper;
    MoveL Offs(pOrigin,195.68,272.14,0.00),v40,z0,tPen\WObj:=wPaper;
    MoveL Offs(pOrigin,195.81,272.66,0.00),v40,z0,tPen\WObj:=wPaper;
    MoveL Offs(pOrigin,201.12,272.66,0.00),v40,fine,tPen\WObj:=wPaper;
    MoveL Offs(pOrigin,201.12,272.66,6.00),v60,z5,tPen\WObj:=wPaper;
    MoveL Offs(pOrigin,198.54,276.58,6.00),vTravel,z5,tPen\WObj:=wPaper;
    MoveL Offs(pOrigin,198.54,276.58,0.00),v60,z0,tPen\WObj:=wPaper;
    MoveL Offs(pOrigin,198.54,278.06,0.00),v40,fine,tPen\WObj:=wPaper;
    MoveL Offs(pOrigin,198.54,278.06,6.00),v60,z5,tPen\WObj:=wPaper;
    MoveL Offs(pOrigin,196.88,276.36,6.00),vTravel,z5,tPen\WObj:=wPaper;
    MoveL Offs(pOrigin,196.88,276.36,0.00),v60,z0,tPen\WObj:=wPaper;
    MoveL Offs(pOrigin,195.60,276.58,0.00),v40,z0,tPen\WObj:=wPaper;
    MoveL Offs(pOrigin,196.43,276.36,0.00),v40,z0,tPen\WObj:=wPaper;
    MoveL Offs(pOrigin,196.43,272.32,0.00),v40,fine,tPen\WObj:=wPaper;
    MoveL Offs(pOrigin,196.43,272.32,6.00),v60,z5,tPen\WObj:=wPaper;
    MoveL Offs(pOrigin,195.09,273.04,6.00),vTravel,z5,tPen\WObj:=wPaper;
    MoveL Offs(pOrigin,195.09,273.04,0.00),v60,z0,tPen\WObj:=wPaper;
    MoveL Offs(pOrigin,204.55,282.50,0.00),v40,z0,tPen\WObj:=wPaper;
    MoveL Offs(pOrigin,205.09,282.01,0.00),v40,z0,tPen\WObj:=wPaper;
    MoveL Offs(pOrigin,189.02,298.08,0.00),v40,fine,tPen\WObj:=wPaper;
    MoveL Offs(pOrigin,189.02,298.08,6.00),v60,z5,tPen\WObj:=wPaper;
    MoveL Offs(pOrigin,189.31,299.28,6.00),vTravel,z5,tPen\WObj:=wPaper;
    MoveL Offs(pOrigin,189.31,299.28,0.00),v60,z0,tPen\WObj:=wPaper;
    MoveL Offs(pOrigin,205.24,283.35,0.00),v40,z0,tPen\WObj:=wPaper;
    MoveL Offs(pOrigin,204.10,283.22,0.00),v40,z0,tPen\WObj:=wPaper;
    MoveL Offs(pOrigin,197.94,283.22,0.00),v40,fine,tPen\WObj:=wPaper;
    MoveL Offs(pOrigin,197.94,283.22,6.00),v60,z5,tPen\WObj:=wPaper;
    MoveL Offs(pOrigin,197.49,281.89,6.00),vTravel,z5,tPen\WObj:=wPaper;
    MoveL Offs(pOrigin,197.49,281.89,0.00),v60,z0,tPen\WObj:=wPaper;
    MoveL Offs(pOrigin,197.49,280.61,0.00),v40,fine,tPen\WObj:=wPaper;
    MoveL Offs(pOrigin,197.49,280.61,6.00),v60,z5,tPen\WObj:=wPaper;
    MoveL Offs(pOrigin,196.43,281.25,6.00),vTravel,z5,tPen\WObj:=wPaper;
    MoveL Offs(pOrigin,196.43,281.25,0.00),v60,z0,tPen\WObj:=wPaper;
    MoveL Offs(pOrigin,196.43,279.76,0.00),v40,fine,tPen\WObj:=wPaper;
    MoveL Offs(pOrigin,196.43,279.76,6.00),v60,z5,tPen\WObj:=wPaper;
    MoveL Offs(pOrigin,200.06,280.06,6.00),vTravel,z5,tPen\WObj:=wPaper;
    MoveL Offs(pOrigin,200.06,280.06,0.00),v60,z0,tPen\WObj:=wPaper;
    MoveL Offs(pOrigin,203.68,280.06,0.00),v40,z0,tPen\WObj:=wPaper;
    MoveL Offs(pOrigin,203.68,281.11,0.00),v40,z0,tPen\WObj:=wPaper;
    MoveL Offs(pOrigin,200.70,281.11,0.00),v40,z0,tPen\WObj:=wPaper;
    MoveL Offs(pOrigin,201.71,281.04,0.00),v40,z0,tPen\WObj:=wPaper;
    MoveL Offs(pOrigin,201.71,282.74,0.00),v40,z0,tPen\WObj:=wPaper;
    MoveL Offs(pOrigin,201.34,283.38,0.00),v40,z0,tPen\WObj:=wPaper;
    MoveL Offs(pOrigin,201.55,283.80,0.00),v40,z0,tPen\WObj:=wPaper;
    MoveL Offs(pOrigin,201.34,283.38,0.00),v40,fine,tPen\WObj:=wPaper;
    MoveL Offs(pOrigin,201.34,283.38,6.00),v60,z5,tPen\WObj:=wPaper;
    MoveL Offs(pOrigin,200.91,282.17,6.00),vTravel,z5,tPen\WObj:=wPaper;
    MoveL Offs(pOrigin,200.91,282.17,0.00),v60,z0,tPen\WObj:=wPaper;
    MoveL Offs(pOrigin,203.89,282.17,0.00),v40,fine,tPen\WObj:=wPaper;
    MoveL Offs(pOrigin,203.89,282.17,6.00),v60,z5,tPen\WObj:=wPaper;
    MoveL Offs(pOrigin,194.96,273.17,6.00),vTravel,z5,tPen\WObj:=wPaper;
    MoveL Offs(pOrigin,194.96,273.17,0.00),v60,z0,tPen\WObj:=wPaper;
    MoveL Offs(pOrigin,194.75,273.60,0.00),v40,z0,tPen\WObj:=wPaper;
  ENDPROC

